LIN {X 0.030,Y -214.228,Z 1696.200,A 0.000,B 0.000,C 90.000,E1 35.931} C_DIS
LIN {X -0.002,Y -206.869,Z 1696.182,A 0.000,B 0.000,C 90.000,E1 32.801} C_DIS
LIN {X -0.016,Y -200.168,Z 1696.165,A 0.000,B 0.000,C 90.000,E1 29.617} C_DIS
LIN {X 0.061,Y -194.075,Z 1696.146,A 0.000,B 0.000,C 90.000,E1 26.360} C_DIS
LIN {X 0.072,Y -188.561,Z 1696.128,A 0.000,B 0.000,C 90.000,E1 23.078} C_DIS
LIN {X 0.078,Y -183.619,Z 1696.110,A 0.000,B 0.000,C 90.000,E1 19.758} C_DIS
LIN {X -0.045,Y -179.365,Z 1696.091,A 0.000,B 0.000,C 90.000,E1 16.441} C_DIS
LIN {X -0.073,Y -175.796,Z 1696.072,A 0.000,B 0.000,C 90.000,E1 13.063} C_DIS
LIN {X -0.080,Y -171.726,Z 1696.044,A 0.000,B 0.000,C 90.000,E1 7.936} C_DIS
LIN {X -0.053,Y -168.927,Z 1696.015,A 0.000,B 0.000,C 90.000,E1 2.751} C_DIS
LIN {X 0.075,Y -168.953,Z 1695.925,A 0.000,B 0.000,C 90.000,E1 346.464} C_DIS
LIN {X 0.065,Y -171.633,Z 1695.896,A 0.000,B 0.000,C 90.000,E1 341.275} C_DIS
LIN {X 0.068,Y -175.125,Z 1695.872,A 0.000,B 0.000,C 90.000,E1 336.975} C_DIS
LIN {X -0.029,Y -179.735,Z 1695.849,A 0.000,B 0.000,C 90.000,E1 332.743} C_DIS
LIN {X 0.084,Y -184.287,Z 1695.830,A 0.000,B 0.000,C 90.000,E1 329.331} C_DIS
LIN {X 0.045,Y -188.356,Z 1695.816,A 0.000,B 0.000,C 90.000,E1 326.834} C_DIS
LIN {X -0.013,Y -194.798,Z 1695.797,A 0.000,B 0.000,C 90.000,E1 323.543} C_DIS
LIN {X 0.017,Y -201.344,Z 1695.782,A 0.000,B 0.000,C 90.000,E1 320.678} C_DIS
LIN {X -0.010,Y -208.807,Z 1695.766,A 0.000,B 0.000,C 90.000,E1 317.877} C_DIS
LIN {X 0.119,Y -217.330,Z 1695.751,A 0.000,B 0.000,C 90.000,E1 315.081} C_DIS
LIN {X -0.014,Y -227.012,Z 1695.736,A 0.000,B 0.000,C 90.000,E1 312.405} C_DIS
LIN {X 0.124,Y -236.194,Z 1695.723,A 0.000,B 0.000,C 90.000,E1 310.092} C_DIS
LIN {X -0.018,Y -246.606,Z 1695.710,A 0.000,B 0.000,C 90.000,E1 307.890} C_DIS
LIN {X -0.140,Y -256.208,Z 1695.700,A 0.000,B 0.000,C 90.000,E1 306.091} C_DIS
LIN {X -0.025,Y -273.225,Z 1695.684,A 0.000,B 0.000,C 90.000,E1 303.214} C_DIS
LIN {X -0.060,Y -291.925,Z 1695.669,A 0.000,B 0.000,C 90.000,E1 300.463} C_DIS
LIN {X 0.104,Y -311.752,Z 1695.654,A 0.000,B 0.000,C 90.000,E1 297.769} C_DIS
LIN {X 0.030,Y -326.865,Z 1695.644,A 0.000,B 0.000,C 90.000,E1 295.848} C_DIS
LIN {X 0.100,Y -342.113,Z 1695.633,A 0.000,B 0.000,C 90.000,E1 293.951} C_DIS
LIN {X -0.138,Y -357.480,Z 1695.623,A 0.000,B 0.000,C 90.000,E1 292.153} C_DIS
LIN {X 0.084,Y -367.403,Z 1695.616,A 0.000,B 0.000,C 90.000,E1 290.918} C_DIS
LIN {X -0.082,Y -374.465,Z 1695.611,A 0.000,B 0.000,C 90.000,E1 290.066} C_DIS
LIN {X 0.242,Y -381.087,Z 1695.607,A 0.000,B 0.000,C 90.000,E1 289.141} C_DIS
LIN {X 0.012,Y -387.016,Z 1695.602,A 0.000,B 0.000,C 90.000,E1 288.308} C_DIS
LIN {X -0.191,Y -390.463,Z 1695.599,A 0.000,B 0.000,C 90.000,E1 287.764} C_DIS
LIN {X 0.165,Y -394.822,Z 1695.594,A 0.000,B 0.000,C 90.000,E1 286.858} C_DIS
LIN {X 0.065,Y -398.245,Z 1695.589,A 0.000,B 0.000,C 90.000,E1 286.024} C_DIS
LIN {X -0.074,Y -400.085,Z 1695.586,A 0.000,B 0.000,C 90.000,E1 285.481} C_DIS
LIN {X 0.072,Y -401.550,Z 1695.583,A 0.000,B 0.000,C 90.000,E1 284.898} C_DIS
LIN {X -0.054,Y -402.648,Z 1695.580,A 0.000,B 0.000,C 90.000,E1 284.356} C_DIS
LIN {X 0.117,Y -403.347,Z 1695.577,A 0.000,B 0.000,C 90.000,E1 283.772} C_DIS
LIN {X -0.094,Y -403.638,Z 1695.573,A 0.000,B 0.000,C 90.000,E1 283.244} C_DIS
LIN {X 0.182,Y -403.524,Z 1695.570,A 0.000,B 0.000,C 90.000,E1 282.647} C_DIS
LIN {X -0.024,Y -402.949,Z 1695.567,A 0.000,B 0.000,C 90.000,E1 282.119} C_DIS
LIN {X 0.163,Y -401.886,Z 1695.564,A 0.000,B 0.000,C 90.000,E1 281.535} C_DIS
LIN {X -0.048,Y -400.295,Z 1695.561,A 0.000,B 0.000,C 90.000,E1 281.007} C_DIS
LIN {X 0.055,Y -398.253,Z 1695.558,A 0.000,B 0.000,C 90.000,E1 280.433} C_DIS
LIN {X -0.169,Y -395.628,Z 1695.555,A 0.000,B 0.000,C 90.000,E1 279.905} C_DIS
LIN {X 0.037,Y -390.912,Z 1695.550,A 0.000,B 0.000,C 90.000,E1 279.029} C_DIS
LIN {X 0.178,Y -383.721,Z 1695.544,A 0.000,B 0.000,C 90.000,E1 277.871} C_DIS
LIN {X -0.205,Y -377.617,Z 1695.539,A 0.000,B 0.000,C 90.000,E1 277.068} C_DIS
LIN {X 0.194,Y -372.861,Z 1695.536,A 0.000,B 0.000,C 90.000,E1 276.429} C_DIS
LIN {X 0.146,Y -367.523,Z 1695.533,A 0.000,B 0.000,C 90.000,E1 275.853} C_DIS
LIN {X -0.105,Y -361.689,Z 1695.530,A 0.000,B 0.000,C 90.000,E1 275.334} C_DIS
LIN {X -0.096,Y -355.702,Z 1695.527,A 0.000,B 0.000,C 90.000,E1 274.821} C_DIS
LIN {X -0.140,Y -349.396,Z 1695.524,A 0.000,B 0.000,C 90.000,E1 274.359} C_DIS
LIN {X -0.004,Y -339.856,Z 1695.521,A 0.000,B 0.000,C 90.000,E1 273.726} C_DIS
LIN {X -0.104,Y -329.964,Z 1695.518,A 0.000,B 0.000,C 90.000,E1 273.212} C_DIS
LIN {X -0.070,Y -320.129,Z 1695.515,A 0.000,B 0.000,C 90.000,E1 272.751} C_DIS
LIN {X -0.097,Y -309.761,Z 1695.513,A 0.000,B 0.000,C 90.000,E1 272.350} C_DIS
LIN {X 0.055,Y -296.182,Z 1695.511,A 0.000,B 0.000,C 90.000,E1 271.892} C_DIS
LIN {X 0.143,Y -285.442,Z 1695.509,A 0.000,B 0.000,C 90.000,E1 271.604} C_DIS
LIN {X -0.086,Y -273.014,Z 1695.508,A 0.000,B 0.000,C 90.000,E1 271.432} C_DIS
LIN {X -0.108,Y -263.030,Z 1695.507,A 0.000,B 0.000,C 90.000,E1 271.318} C_DIS
LIN {X 0.113,Y -249.683,Z 1695.507,A 0.000,B 0.000,C 90.000,E1 271.203} C_DIS
LIN {X 0.064,Y -190.443,Z 1695.507,A 0.000,B 0.000,C 90.000,E1 271.203} C_DIS
LIN {X -0.003,Y -184.503,Z 1695.507,A 0.000,B 0.000,C 90.000,E1 271.203} C_DIS
LIN {X -0.024,Y -181.413,Z 1695.507,A 0.000,B 0.000,C 90.000,E1 271.203} C_DIS
LIN {X 0.029,Y -181.579,Z 1695.501,A 0.000,B 0.000,C 90.000,E1 270.172} C_DIS
LIN {X 0.033,Y -180.853,Z 1695.472,A 0.000,B 0.000,C 90.000,E1 264.951} C_DIS
LIN {X -0.062,Y -178.964,Z 1695.444,A 0.000,B 0.000,C 90.000,E1 259.916} C_DIS
LIN {X 0.006,Y -177.372,Z 1695.430,A 0.000,B 0.000,C 90.000,E1 257.353} C_DIS
LIN {X -0.067,Y -175.547,Z 1695.411,A 0.000,B 0.000,C 90.000,E1 253.976} C_DIS
LIN {X -0.059,Y -172.279,Z 1695.387,A 0.000,B 0.000,C 90.000,E1 249.699} C_DIS
LIN {X -0.020,Y -171.758,Z 1695.382,A 0.000,B 0.000,C 90.000,E1 248.827} C_DIS
LIN {X -0.003,Y -167.358,Z 1695.354,A 0.000,B 0.000,C 90.000,E1 243.640} C_DIS
LIN {X 0.080,Y -166.747,Z 1695.349,A 0.000,B 0.000,C 90.000,E1 242.743} C_DIS
LIN {X -0.009,Y -162.727,Z 1695.324,A 0.000,B 0.000,C 90.000,E1 238.408} C_DIS
LIN {X 0.052,Y -161.417,Z 1695.315,A 0.000,B 0.000,C 90.000,E1 236.628} C_DIS
LIN {X 0.094,Y -157.409,Z 1695.290,A 0.000,B 0.000,C 90.000,E1 232.190} C_DIS
LIN {X 0.027,Y -155.411,Z 1695.275,A 0.000,B 0.000,C 90.000,E1 229.542} C_DIS
LIN {X -0.042,Y -151.740,Z 1695.250,A 0.000,B 0.000,C 90.000,E1 225.081} C_DIS
LIN {X -0.030,Y -149.937,Z 1695.235,A 0.000,B 0.000,C 90.000,E1 222.366} C_DIS
LIN {X -0.002,Y -146.785,Z 1695.210,A 0.000,B 0.000,C 90.000,E1 217.810} C_DIS
LIN {X -0.018,Y -145.357,Z 1695.195,A 0.000,B 0.000,C 90.000,E1 215.072} C_DIS
LIN {X 0.016,Y -142.427,Z 1695.164,A 0.000,B 0.000,C 90.000,E1 209.539} C_DIS
LIN {X 0.064,Y -141.415,Z 1695.149,A 0.000,B 0.000,C 90.000,E1 206.744} C_DIS
LIN {X 0.052,Y -139.361,Z 1695.113,A 0.000,B 0.000,C 90.000,E1 200.248} C_DIS
LIN {X 0.039,Y -138.803,Z 1695.097,A 0.000,B 0.000,C 90.000,E1 197.457} C_DIS
LIN {X -0.042,Y -138.349,Z 1695.056,A 0.000,B 0.000,C 90.000,E1 190.018} C_DIS
LIN {X -0.027,Y -139.365,Z 1695.009,A 0.000,B 0.000,C 90.000,E1 181.604} C_DIS
LIN {X 0.026,Y -141.250,Z 1694.973,A 0.000,B 0.000,C 90.000,E1 175.065} C_DIS
LIN {X -0.016,Y -142.619,Z 1694.957,A 0.000,B 0.000,C 90.000,E1 172.299} C_DIS
LIN {X -0.063,Y -144.938,Z 1694.932,A 0.000,B 0.000,C 90.000,E1 167.701} C_DIS
LIN {X 0.070,Y -147.566,Z 1694.911,A 0.000,B 0.000,C 90.000,E1 163.976} C_DIS
LIN {X -0.040,Y -150.174,Z 1694.891,A 0.000,B 0.000,C 90.000,E1 160.369} C_DIS
LIN {X -0.032,Y -153.551,Z 1694.871,A 0.000,B 0.000,C 90.000,E1 156.741} C_DIS
LIN {X 0.020,Y -156.968,Z 1694.851,A 0.000,B 0.000,C 90.000,E1 153.127} C_DIS
LIN {X -0.045,Y -161.077,Z 1694.831,A 0.000,B 0.000,C 90.000,E1 149.587} C_DIS
LIN {X 0.040,Y -163.184,Z 1694.821,A 0.000,B 0.000,C 90.000,E1 147.788} C_DIS
LIN {X 0.046,Y -167.605,Z 1694.802,A 0.000,B 0.000,C 90.000,E1 144.276} C_DIS
LIN {X -0.045,Y -171.433,Z 1694.787,A 0.000,B 0.000,C 90.000,E1 141.698} C_DIS
LIN {X -0.007,Y -176.354,Z 1694.768,A 0.000,B 0.000,C 90.000,E1 138.243} C_DIS
LIN {X -0.011,Y -180.645,Z 1694.754,A 0.000,B 0.000,C 90.000,E1 135.688} C_DIS
LIN {X -0.026,Y -186.047,Z 1694.735,A 0.000,B 0.000,C 90.000,E1 132.324} C_DIS
LIN {X 0.036,Y -190.683,Z 1694.721,A 0.000,B 0.000,C 90.000,E1 129.806} C_DIS
LIN {X 0.069,Y -196.434,Z 1694.703,A 0.000,B 0.000,C 90.000,E1 126.503} C_DIS
LIN {X 0.037,Y -201.219,Z 1694.689,A 0.000,B 0.000,C 90.000,E1 124.072} C_DIS
LIN {X 0.048,Y -207.544,Z 1694.670,A 0.000,B 0.000,C 90.000,E1 120.669} C_DIS
LIN {X 0.007,Y -208.682,Z 1694.667,A 0.000,B 0.000,C 90.000,E1 120.129} C_DIS
LIN {X -0.025,Y -331.531,Z 1694.667,A 0.000,B 0.000,C 90.000,E1 120.129} C_DIS
LIN {X -0.066,Y -334.422,Z 1694.667,A 0.000,B 0.000,C 90.000,E1 120.079} C_DIS
LIN {X 0.082,Y -337.325,Z 1694.666,A 0.000,B 0.000,C 90.000,E1 119.922} C_DIS
LIN {X -0.059,Y -340.923,Z 1694.665,A 0.000,B 0.000,C 90.000,E1 119.667} C_DIS
LIN {X 0.003,Y -344.532,Z 1694.662,A 0.000,B 0.000,C 90.000,E1 119.205} C_DIS
LIN {X -0.009,Y -346.257,Z 1694.661,A 0.000,B 0.000,C 90.000,E1 118.899} C_DIS
LIN {X 0.097,Y -360.412,Z 1694.644,A 0.000,B 0.000,C 90.000,E1 115.848} C_DIS
LIN {X -0.077,Y -374.699,Z 1694.629,A 0.000,B 0.000,C 90.000,E1 113.206} C_DIS
LIN {X 0.067,Y -388.768,Z 1694.616,A 0.000,B 0.000,C 90.000,E1 110.865} C_DIS
LIN {X 0.061,Y -404.224,Z 1694.603,A 0.000,B 0.000,C 90.000,E1 108.598} C_DIS
LIN {X 0.046,Y -421.177,Z 1694.591,A 0.000,B 0.000,C 90.000,E1 106.386} C_DIS
LIN {X -0.074,Y -439.740,Z 1694.579,A 0.000,B 0.000,C 90.000,E1 104.245} C_DIS
LIN {X -0.046,Y -459.590,Z 1694.568,A 0.000,B 0.000,C 90.000,E1 102.187} C_DIS
LIN {X -0.042,Y -482.573,Z 1694.556,A 0.000,B 0.000,C 90.000,E1 100.074} C_DIS
LIN {X 0.077,Y -503.529,Z 1694.546,A 0.000,B 0.000,C 90.000,E1 98.341} C_DIS
LIN {X -0.170,Y -505.736,Z 1694.545,A 0.000,B 0.000,C 90.000,E1 98.163} C_DIS
LIN {X -0.204,Y -507.593,Z 1694.544,A 0.000,B 0.000,C 90.000,E1 97.936} C_DIS
LIN {X -0.168,Y -508.999,Z 1694.543,A 0.000,B 0.000,C 90.000,E1 97.701} C_DIS
LIN {X 0.164,Y -510.872,Z 1694.540,A 0.000,B 0.000,C 90.000,E1 97.182} C_DIS
LIN {X 0.000,Y -511.603,Z 1694.537,A 0.000,B 0.000,C 90.000,E1 96.720} C_DIS
LIN {X -0.155,Y -511.316,Z 1694.535,A 0.000,B 0.000,C 90.000,E1 96.258} C_DIS
LIN {X 0.201,Y -509.964,Z 1694.532,A 0.000,B 0.000,C 90.000,E1 95.739} C_DIS
LIN {X 0.100,Y -508.818,Z 1694.531,A 0.000,B 0.000,C 90.000,E1 95.511} C_DIS
LIN {X -0.059,Y -505.504,Z 1694.528,A 0.000,B 0.000,C 90.000,E1 95.049} C_DIS
LIN {X -0.182,Y -494.848,Z 1694.520,A 0.000,B 0.000,C 90.000,E1 93.612} C_DIS
LIN {X -0.020,Y -484.051,Z 1694.512,A 0.000,B 0.000,C 90.000,E1 92.121} C_DIS
LIN {X -0.222,Y -471.379,Z 1694.502,A 0.000,B 0.000,C 90.000,E1 90.401} C_DIS
LIN {X 0.000,Y -460.498,Z 1694.494,A 0.000,B 0.000,C 90.000,E1 88.854} C_DIS
LIN {X 0.036,Y -449.452,Z 1694.485,A 0.000,B 0.000,C 90.000,E1 87.306} C_DIS
LIN {X -0.089,Y -438.224,Z 1694.476,A 0.000,B 0.000,C 90.000,E1 85.755} C_DIS
LIN {X 0.191,Y -424.959,Z 1694.466,A 0.000,B 0.000,C 90.000,E1 83.856} C_DIS
LIN {X 0.022,Y -408.389,Z 1694.452,A 0.000,B 0.000,C 90.000,E1 81.432} C_DIS
LIN {X 0.199,Y -387.530,Z 1694.434,A 0.000,B 0.000,C 90.000,E1 78.049} C_DIS
LIN {X 0.168,Y -374.325,Z 1694.421,A 0.000,B 0.000,C 90.000,E1 75.755} C_DIS
LIN {X 0.016,Y -361.481,Z 1694.408,A 0.000,B 0.000,C 90.000,E1 73.433} C_DIS
LIN {X 0.064,Y -345.943,Z 1694.391,A 0.000,B 0.000,C 90.000,E1 70.423} C_DIS
LIN {X -0.014,Y -331.397,Z 1694.374,A 0.000,B 0.000,C 90.000,E1 67.358} C_DIS
LIN {X -0.093,Y -318.829,Z 1694.358,A 0.000,B 0.000,C 90.000,E1 64.537} C_DIS
LIN {X -0.097,Y -306.555,Z 1694.342,A 0.000,B 0.000,C 90.000,E1 61.641} C_DIS
LIN {X -0.046,Y -298.534,Z 1694.331,A 0.000,B 0.000,C 90.000,E1 59.665} C_DIS
LIN {X -0.009,Y -288.988,Z 1694.318,A 0.000,B 0.000,C 90.000,E1 57.327} C_DIS
LIN {X -0.069,Y -280.700,Z 1694.307,A 0.000,B 0.000,C 90.000,E1 55.308} C_DIS
LIN {X 0.104,Y -272.100,Z 1694.296,A 0.000,B 0.000,C 90.000,E1 53.210} C_DIS
LIN {X -0.089,Y -262.186,Z 1694.282,A 0.000,B 0.000,C 90.000,E1 50.803} C_DIS
LIN {X 0.009,Y -252.457,Z 1694.268,A 0.000,B 0.000,C 90.000,E1 48.286} C_DIS
LIN {X 0.037,Y -240.583,Z 1694.250,A 0.000,B 0.000,C 90.000,E1 45.000} C_DIS
LIN {X -0.055,Y -230.918,Z 1694.234,A 0.000,B 0.000,C 90.000,E1 42.043} C_DIS
LIN {X -0.002,Y -222.030,Z 1694.217,A 0.000,B 0.000,C 90.000,E1 38.991} C_DIS
LIN {X 0.072,Y -214.005,Z 1694.199,A 0.000,B 0.000,C 90.000,E1 35.884} C_DIS
LIN {X 0.041,Y -206.678,Z 1694.182,A 0.000,B 0.000,C 90.000,E1 32.752} C_DIS
LIN {X -0.048,Y -200.026,Z 1694.164,A 0.000,B 0.000,C 90.000,E1 29.589} C_DIS
LIN {X -0.070,Y -193.968,Z 1694.146,A 0.000,B 0.000,C 90.000,E1 26.360} C_DIS
LIN {X -0.058,Y -188.449,Z 1694.128,A 0.000,B 0.000,C 90.000,E1 23.078} C_DIS
LIN {X -0.052,Y -183.528,Z 1694.110,A 0.000,B 0.000,C 90.000,E1 19.758} C_DIS
LIN {X -0.001,Y -179.277,Z 1694.091,A 0.000,B 0.000,C 90.000,E1 16.386} C_DIS
LIN {X -0.030,Y -175.708,Z 1694.072,A 0.000,B 0.000,C 90.000,E1 13.008} C_DIS
LIN {X -0.064,Y -172.241,Z 1694.048,A 0.000,B 0.000,C 90.000,E1 8.746} C_DIS
LIN {X -0.002,Y -169.206,Z 1694.020,A 0.000,B 0.000,C 90.000,E1 3.555} C_DIS
LIN {X 0.014,Y -167.284,Z 1693.973,A 0.000,B 0.000,C 90.000,E1 355.179} C_DIS
LIN {X 0.070,Y -168.897,Z 1693.925,A 0.000,B 0.000,C 90.000,E1 346.464} C_DIS
LIN {X 0.056,Y -171.617,Z 1693.896,A 0.000,B 0.000,C 90.000,E1 341.275} C_DIS
LIN {X 0.059,Y -175.114,Z 1693.872,A 0.000,B 0.000,C 90.000,E1 336.975} C_DIS
LIN {X -0.038,Y -179.765,Z 1693.849,A 0.000,B 0.000,C 90.000,E1 332.743} C_DIS
LIN {X 0.076,Y -184.359,Z 1693.830,A 0.000,B 0.000,C 90.000,E1 329.331} C_DIS
LIN {X 0.037,Y -188.457,Z 1693.816,A 0.000,B 0.000,C 90.000,E1 326.834} C_DIS
LIN {X -0.018,Y -194.926,Z 1693.797,A 0.000,B 0.000,C 90.000,E1 323.543} C_DIS
LIN {X 0.015,Y -201.480,Z 1693.782,A 0.000,B 0.000,C 90.000,E1 320.678} C_DIS
LIN {X -0.009,Y -208.972,Z 1693.766,A 0.000,B 0.000,C 90.000,E1 317.877} C_DIS
LIN {X -0.030,Y -217.522,Z 1693.751,A 0.000,B 0.000,C 90.000,E1 315.121} C_DIS
LIN {X -0.005,Y -227.218,Z 1693.736,A 0.000,B 0.000,C 90.000,E1 312.405} C_DIS
LIN {X 0.138,Y -236.411,Z 1693.723,A 0.000,B 0.000,C 90.000,E1 310.092} C_DIS
LIN {X 0.001,Y -246.816,Z 1693.710,A 0.000,B 0.000,C 90.000,E1 307.890} C_DIS
LIN {X -0.117,Y -256.413,Z 1693.700,A 0.000,B 0.000,C 90.000,E1 306.091} C_DIS
LIN {X 0.004,Y -273.378,Z 1693.685,A 0.000,B 0.000,C 90.000,E1 303.214} C_DIS
LIN {X -0.025,Y -292.060,Z 1693.669,A 0.000,B 0.000,C 90.000,E1 300.463} C_DIS
LIN {X 0.145,Y -311.848,Z 1693.654,A 0.000,B 0.000,C 90.000,E1 297.769} C_DIS
LIN {X 0.075,Y -326.940,Z 1693.644,A 0.000,B 0.000,C 90.000,E1 295.848} C_DIS
LIN {X 0.148,Y -342.149,Z 1693.633,A 0.000,B 0.000,C 90.000,E1 293.951} C_DIS
LIN {X -0.088,Y -357.514,Z 1693.623,A 0.000,B 0.000,C 90.000,E1 292.153} C_DIS
LIN {X 0.137,Y -367.416,Z 1693.616,A 0.000,B 0.000,C 90.000,E1 290.918} C_DIS
LIN {X -0.092,Y -374.554,Z 1693.611,A 0.000,B 0.000,C 90.000,E1 290.066} C_DIS
LIN {X 0.232,Y -381.182,Z 1693.607,A 0.000,B 0.000,C 90.000,E1 289.141} C_DIS
LIN {X 0.004,Y -387.101,Z 1693.602,A 0.000,B 0.000,C 90.000,E1 288.308} C_DIS
LIN {X -0.199,Y -390.540,Z 1693.599,A 0.000,B 0.000,C 90.000,E1 287.764} C_DIS
LIN {X 0.157,Y -394.932,Z 1693.594,A 0.000,B 0.000,C 90.000,E1 286.858} C_DIS
LIN {X 0.059,Y -398.389,Z 1693.589,A 0.000,B 0.000,C 90.000,E1 286.024} C_DIS
LIN {X -0.080,Y -400.222,Z 1693.586,A 0.000,B 0.000,C 90.000,E1 285.481} C_DIS
LIN {X 0.067,Y -401.679,Z 1693.583,A 0.000,B 0.000,C 90.000,E1 284.898} C_DIS
LIN {X -0.059,Y -402.830,Z 1693.580,A 0.000,B 0.000,C 90.000,E1 284.356} C_DIS
LIN {X 0.114,Y -403.515,Z 1693.577,A 0.000,B 0.000,C 90.000,E1 283.772} C_DIS
LIN {X -0.096,Y -403.833,Z 1693.573,A 0.000,B 0.000,C 90.000,E1 283.244} C_DIS
LIN {X 0.182,Y -403.732,Z 1693.570,A 0.000,B 0.000,C 90.000,E1 282.647} C_DIS
LIN {X -0.024,Y -403.154,Z 1693.567,A 0.000,B 0.000,C 90.000,E1 282.119} C_DIS
LIN {X 0.164,Y -402.104,Z 1693.564,A 0.000,B 0.000,C 90.000,E1 281.535} C_DIS
LIN {X -0.046,Y -400.527,Z 1693.561,A 0.000,B 0.000,C 90.000,E1 281.007} C_DIS
LIN {X 0.058,Y -398.464,Z 1693.558,A 0.000,B 0.000,C 90.000,E1 280.433} C_DIS
LIN {X -0.165,Y -395.866,Z 1693.555,A 0.000,B 0.000,C 90.000,E1 279.905} C_DIS
LIN {X 0.044,Y -391.171,Z 1693.550,A 0.000,B 0.000,C 90.000,E1 279.029} C_DIS
LIN {X 0.150,Y -385.815,Z 1693.545,A 0.000,B 0.000,C 90.000,E1 278.163} C_DIS
LIN {X -0.175,Y -379.906,Z 1693.541,A 0.000,B 0.000,C 90.000,E1 277.352} C_DIS
LIN {X -0.178,Y -375.435,Z 1693.537,A 0.000,B 0.000,C 90.000,E1 276.777} C_DIS
LIN {X 0.164,Y -370.366,Z 1693.534,A 0.000,B 0.000,C 90.000,E1 276.144} C_DIS
LIN {X -0.150,Y -364.742,Z 1693.531,A 0.000,B 0.000,C 90.000,E1 275.625} C_DIS
LIN {X 0.139,Y -358.847,Z 1693.528,A 0.000,B 0.000,C 90.000,E1 275.049} C_DIS
LIN {X -0.023,Y -352.666,Z 1693.526,A 0.000,B 0.000,C 90.000,E1 274.588} C_DIS
LIN {X 0.048,Y -346.231,Z 1693.523,A 0.000,B 0.000,C 90.000,E1 274.131} C_DIS
LIN {X 0.067,Y -339.748,Z 1693.521,A 0.000,B 0.000,C 90.000,E1 273.726} C_DIS
LIN {X -0.040,Y -329.761,Z 1693.518,A 0.000,B 0.000,C 90.000,E1 273.212} C_DIS
LIN {X -0.023,Y -319.765,Z 1693.515,A 0.000,B 0.000,C 90.000,E1 272.751} C_DIS
LIN {X 0.050,Y -313.001,Z 1693.514,A 0.000,B 0.000,C 90.000,E1 272.465} C_DIS
LIN {X -0.019,Y -302.463,Z 1693.512,A 0.000,B 0.000,C 90.000,E1 272.121} C_DIS
LIN {X -0.068,Y -292.250,Z 1693.510,A 0.000,B 0.000,C 90.000,E1 271.835} C_DIS
LIN {X 0.100,Y -280.775,Z 1693.509,A 0.000,B 0.000,C 90.000,E1 271.547} C_DIS
LIN {X -0.023,Y -268.128,Z 1693.508,A 0.000,B 0.000,C 90.000,E1 271.375} C_DIS
LIN {X 0.128,Y -259.488,Z 1693.507,A 0.000,B 0.000,C 90.000,E1 271.260} C_DIS
LIN {X -0.001,Y -250.689,Z 1693.507,A 0.000,B 0.000,C 90.000,E1 271.260} C_DIS
LIN {X -0.023,Y -196.001,Z 1693.507,A 0.000,B 0.000,C 90.000,E1 271.260} C_DIS
LIN {X 0.038,Y -186.326,Z 1693.507,A 0.000,B 0.000,C 90.000,E1 271.203} C_DIS
LIN {X 0.001,Y -181.411,Z 1693.507,A 0.000,B 0.000,C 90.000,E1 271.203} C_DIS
LIN {X -0.015,Y -181.581,Z 1693.502,A 0.000,B 0.000,C 90.000,E1 270.286} C_DIS
LIN {X -0.040,Y -180.899,Z 1693.474,A 0.000,B 0.000,C 90.000,E1 265.241} C_DIS
LIN {X -0.091,Y -180.211,Z 1693.464,A 0.000,B 0.000,C 90.000,E1 263.571} C_DIS
LIN {X 0.039,Y -179.033,Z 1693.445,A 0.000,B 0.000,C 90.000,E1 260.151} C_DIS
LIN {X -0.074,Y -178.686,Z 1693.441,A 0.000,B 0.000,C 90.000,E1 259.342} C_DIS
LIN {X 0.037,Y -175.736,Z 1693.412,A 0.000,B 0.000,C 90.000,E1 254.212} C_DIS
LIN {X 0.033,Y -171.920,Z 1693.384,A 0.000,B 0.000,C 90.000,E1 249.082} C_DIS
LIN {X 0.007,Y -171.291,Z 1693.379,A 0.000,B 0.000,C 90.000,E1 248.230} C_DIS
LIN {X 0.053,Y -167.556,Z 1693.355,A 0.000,B 0.000,C 90.000,E1 243.896} C_DIS
LIN {X 0.067,Y -166.179,Z 1693.345,A 0.000,B 0.000,C 90.000,E1 242.153} C_DIS
LIN {X 0.056,Y -162.950,Z 1693.326,A 0.000,B 0.000,C 90.000,E1 238.663} C_DIS
LIN {X 0.103,Y -160.856,Z 1693.311,A 0.000,B 0.000,C 90.000,E1 236.008} C_DIS
LIN {X 0.081,Y -157.633,Z 1693.292,A 0.000,B 0.000,C 90.000,E1 232.477} C_DIS
LIN {X 0.018,Y -155.670,Z 1693.277,A 0.000,B 0.000,C 90.000,E1 229.828} C_DIS
LIN {X 0.071,Y -151.937,Z 1693.252,A 0.000,B 0.000,C 90.000,E1 225.324} C_DIS
LIN {X 0.085,Y -150.175,Z 1693.237,A 0.000,B 0.000,C 90.000,E1 222.609} C_DIS
LIN {X 0.005,Y -146.951,Z 1693.212,A 0.000,B 0.000,C 90.000,E1 218.096} C_DIS
LIN {X -0.007,Y -145.538,Z 1693.196,A 0.000,B 0.000,C 90.000,E1 215.358} C_DIS
LIN {X 0.031,Y -142.935,Z 1693.171,A 0.000,B 0.000,C 90.000,E1 210.747} C_DIS
LIN {X -0.033,Y -141.558,Z 1693.150,A 0.000,B 0.000,C 90.000,E1 207.078} C_DIS
LIN {X 0.020,Y -139.408,Z 1693.114,A 0.000,B 0.000,C 90.000,E1 200.556} C_DIS
LIN {X -0.059,Y -139.128,Z 1693.104,A 0.000,B 0.000,C 90.000,E1 198.725} C_DIS
LIN {X -0.032,Y -138.350,Z 1693.057,A 0.000,B 0.000,C 90.000,E1 190.310} C_DIS
LIN {X -0.044,Y -139.498,Z 1693.005,A 0.000,B 0.000,C 90.000,E1 180.974} C_DIS
LIN {X 0.037,Y -141.121,Z 1692.974,A 0.000,B 0.000,C 90.000,E1 175.355} C_DIS
LIN {X -0.010,Y -142.502,Z 1692.959,A 0.000,B 0.000,C 90.000,E1 172.591} C_DIS
LIN {X -0.064,Y -144.757,Z 1692.933,A 0.000,B 0.000,C 90.000,E1 167.993} C_DIS
LIN {X 0.027,Y -147.368,Z 1692.913,A 0.000,B 0.000,C 90.000,E1 164.283} C_DIS
LIN {X -0.051,Y -150.696,Z 1692.887,A 0.000,B 0.000,C 90.000,E1 159.752} C_DIS
LIN {X 0.032,Y -154.175,Z 1692.867,A 0.000,B 0.000,C 90.000,E1 156.102} C_DIS
LIN {X -0.038,Y -157.611,Z 1692.847,A 0.000,B 0.000,C 90.000,E1 152.538} C_DIS
LIN {X 0.050,Y -161.863,Z 1692.828,A 0.000,B 0.000,C 90.000,E1 148.948} C_DIS
LIN {X -0.071,Y -166.054,Z 1692.808,A 0.000,B 0.000,C 90.000,E1 145.468} C_DIS
LIN {X -0.080,Y -171.059,Z 1692.789,A 0.000,B 0.000,C 90.000,E1 141.984} C_DIS
LIN {X -0.050,Y -175.931,Z 1692.770,A 0.000,B 0.000,C 90.000,E1 138.528} C_DIS
LIN {X -0.058,Y -180.170,Z 1692.755,A 0.000,B 0.000,C 90.000,E1 135.972} C_DIS
LIN {X -0.090,Y -185.587,Z 1692.737,A 0.000,B 0.000,C 90.000,E1 132.609} C_DIS
LIN {X -0.040,Y -190.178,Z 1692.723,A 0.000,B 0.000,C 90.000,E1 130.092} C_DIS
LIN {X 0.005,Y -197.508,Z 1692.700,A 0.000,B 0.000,C 90.000,E1 125.964} C_DIS
LIN {X 0.046,Y -200.776,Z 1692.691,A 0.000,B 0.000,C 90.000,E1 124.326} C_DIS
LIN {X -0.044,Y -206.667,Z 1692.673,A 0.000,B 0.000,C 90.000,E1 121.131} C_DIS
LIN {X -0.036,Y -208.602,Z 1692.668,A 0.000,B 0.000,C 90.000,E1 120.178} C_DIS
LIN {X 0.181,Y -331.416,Z 1692.668,A 0.000,B 0.000,C 90.000,E1 120.129} C_DIS
LIN {X 0.084,Y -332.682,Z 1692.667,A 0.000,B 0.000,C 90.000,E1 120.129} C_DIS
LIN {X -0.072,Y -336.857,Z 1692.667,A 0.000,B 0.000,C 90.000,E1 120.001} C_DIS
LIN {X 0.063,Y -339.147,Z 1692.666,A 0.000,B 0.000,C 90.000,E1 119.823} C_DIS
LIN {X -0.086,Y -342.286,Z 1692.664,A 0.000,B 0.000,C 90.000,E1 119.539} C_DIS
LIN {X -0.111,Y -345.841,Z 1692.661,A 0.000,B 0.000,C 90.000,E1 118.999} C_DIS
LIN {X -0.149,Y -361.491,Z 1692.642,A 0.000,B 0.000,C 90.000,E1 115.668} C_DIS
LIN {X 0.197,Y -375.906,Z 1692.628,A 0.000,B 0.000,C 90.000,E1 112.950} C_DIS
LIN {X 0.012,Y -390.096,Z 1692.615,A 0.000,B 0.000,C 90.000,E1 110.663} C_DIS
LIN {X -0.107,Y -405.685,Z 1692.602,A 0.000,B 0.000,C 90.000,E1 108.417} C_DIS
LIN {X -0.091,Y -422.779,Z 1692.590,A 0.000,B 0.000,C 90.000,E1 106.205} C_DIS
LIN {X -0.180,Y -441.497,Z 1692.578,A 0.000,B 0.000,C 90.000,E1 104.064} C_DIS
LIN {X -0.035,Y -461.400,Z 1692.567,A 0.000,B 0.000,C 90.000,E1 102.007} C_DIS
LIN {X 0.011,Y -484.436,Z 1692.555,A 0.000,B 0.000,C 90.000,E1 99.905} C_DIS
LIN {X 0.059,Y -502.801,Z 1692.547,A 0.000,B 0.000,C 90.000,E1 98.398} C_DIS
LIN {X -0.173,Y -505.121,Z 1692.546,A 0.000,B 0.000,C 90.000,E1 98.219} C_DIS
LIN {X 0.021,Y -506.880,Z 1692.544,A 0.000,B 0.000,C 90.000,E1 97.992} C_DIS
LIN {X -0.037,Y -508.464,Z 1692.543,A 0.000,B 0.000,C 90.000,E1 97.757} C_DIS
LIN {X -0.163,Y -509.645,Z 1692.542,A 0.000,B 0.000,C 90.000,E1 97.530} C_DIS
LIN {X 0.176,Y -511.052,Z 1692.539,A 0.000,B 0.000,C 90.000,E1 97.011} C_DIS
LIN {X 0.017,Y -511.389,Z 1692.536,A 0.000,B 0.000,C 90.000,E1 96.549} C_DIS
LIN {X -0.136,Y -510.711,Z 1692.534,A 0.000,B 0.000,C 90.000,E1 96.087} C_DIS
LIN {X 0.221,Y -508.900,Z 1692.531,A 0.000,B 0.000,C 90.000,E1 95.568} C_DIS
LIN {X 0.166,Y -507.457,Z 1692.530,A 0.000,B 0.000,C 90.000,E1 95.334} C_DIS
LIN {X -0.059,Y -495.068,Z 1692.520,A 0.000,B 0.000,C 90.000,E1 93.669} C_DIS
LIN {X 0.104,Y -484.289,Z 1692.512,A 0.000,B 0.000,C 90.000,E1 92.178} C_DIS
LIN {X -0.102,Y -471.624,Z 1692.502,A 0.000,B 0.000,C 90.000,E1 90.458} C_DIS
LIN {X 0.122,Y -460.741,Z 1692.494,A 0.000,B 0.000,C 90.000,E1 88.912} C_DIS
LIN {X 0.160,Y -449.733,Z 1692.485,A 0.000,B 0.000,C 90.000,E1 87.364} C_DIS
LIN {X 0.206,Y -436.612,Z 1692.475,A 0.000,B 0.000,C 90.000,E1 85.527} C_DIS
LIN {X 0.180,Y -421.443,Z 1692.463,A 0.000,B 0.000,C 90.000,E1 83.394} C_DIS
LIN {X -0.130,Y -406.764,Z 1692.451,A 0.000,B 0.000,C 90.000,E1 81.254} C_DIS
LIN {X -0.073,Y -385.987,Z 1692.433,A 0.000,B 0.000,C 90.000,E1 77.881} C_DIS
LIN {X -0.048,Y -372.788,Z 1692.420,A 0.000,B 0.000,C 90.000,E1 75.574} C_DIS
LIN {X 0.119,Y -359.960,Z 1692.407,A 0.000,B 0.000,C 90.000,E1 73.196} C_DIS
LIN {X 0.112,Y -344.472,Z 1692.390,A 0.000,B 0.000,C 90.000,E1 70.188} C_DIS
LIN {X 0.126,Y -331.422,Z 1692.375,A 0.000,B 0.000,C 90.000,E1 67.411} C_DIS
LIN {X 0.054,Y -318.860,Z 1692.359,A 0.000,B 0.000,C 90.000,E1 64.588} C_DIS
LIN {X 0.048,Y -306.589,Z 1692.343,A 0.000,B 0.000,C 90.000,E1 61.691} C_DIS
LIN {X -0.050,Y -298.566,Z 1692.332,A 0.000,B 0.000,C 90.000,E1 59.744} C_DIS
LIN {X 0.145,Y -289.028,Z 1692.319,A 0.000,B 0.000,C 90.000,E1 57.375} C_DIS
LIN {X -0.073,Y -280.721,Z 1692.308,A 0.000,B 0.000,C 90.000,E1 55.388} C_DIS
LIN {X -0.121,Y -272.130,Z 1692.296,A 0.000,B 0.000,C 90.000,E1 53.336} C_DIS
LIN {X -0.040,Y -260.777,Z 1692.281,A 0.000,B 0.000,C 90.000,E1 50.517} C_DIS
LIN {X 0.024,Y -251.064,Z 1692.267,A 0.000,B 0.000,C 90.000,E1 48.000} C_DIS
LIN {X 0.006,Y -239.326,Z 1692.248,A 0.000,B 0.000,C 90.000,E1 44.717} C_DIS
LIN {X -0.001,Y -228.651,Z 1692.230,A 0.000,B 0.000,C 90.000,E1 41.353} C_DIS
LIN {X 0.071,Y -221.026,Z 1692.215,A 0.000,B 0.000,C 90.000,E1 38.669} C_DIS
LIN {X -0.015,Y -213.117,Z 1692.198,A 0.000,B 0.000,C 90.000,E1 35.598} C_DIS
LIN {X -0.068,Y -205.886,Z 1692.180,A 0.000,B 0.000,C 90.000,E1 32.467} C_DIS
LIN {X -0.102,Y -199.321,Z 1692.162,A 0.000,B 0.000,C 90.000,E1 29.283} C_DIS
LIN {X -0.047,Y -193.335,Z 1692.145,A 0.000,B 0.000,C 90.000,E1 26.027} C_DIS
LIN {X 0.043,Y -187.880,Z 1692.126,A 0.000,B 0.000,C 90.000,E1 22.717} C_DIS
LIN {X 0.036,Y -183.036,Z 1692.108,A 0.000,B 0.000,C 90.000,E1 19.396} C_DIS
LIN {X 0.073,Y -178.843,Z 1692.089,A 0.000,B 0.000,C 90.000,E1 16.024} C_DIS
LIN {X 0.028,Y -175.347,Z 1692.070,A 0.000,B 0.000,C 90.000,E1 12.647} C_DIS
LIN {X -0.054,Y -171.950,Z 1692.047,A 0.000,B 0.000,C 90.000,E1 8.398} C_DIS
LIN {X -0.018,Y -168.990,Z 1692.018,A 0.000,B 0.000,C 90.000,E1 3.212} C_DIS
LIN {X 0.013,Y -167.228,Z 1691.973,A 0.000,B 0.000,C 90.000,E1 355.179} C_DIS
LIN {X 0.064,Y -168.855,Z 1691.925,A 0.000,B 0.000,C 90.000,E1 346.464} C_DIS
LIN {X 0.049,Y -171.597,Z 1691.896,A 0.000,B 0.000,C 90.000,E1 341.275} C_DIS
LIN {X 0.051,Y -175.105,Z 1691.872,A 0.000,B 0.000,C 90.000,E1 336.975} C_DIS
LIN {X -0.047,Y -179.803,Z 1691.849,A 0.000,B 0.000,C 90.000,E1 332.743} C_DIS
LIN {X 0.069,Y -184.434,Z 1691.830,A 0.000,B 0.000,C 90.000,E1 329.331} C_DIS
LIN {X 0.032,Y -188.559,Z 1691.816,A 0.000,B 0.000,C 90.000,E1 326.834} C_DIS
LIN {X -0.022,Y -195.053,Z 1691.797,A 0.000,B 0.000,C 90.000,E1 323.543} C_DIS
LIN {X 0.014,Y -201.616,Z 1691.782,A 0.000,B 0.000,C 90.000,E1 320.678} C_DIS
LIN {X -0.008,Y -209.137,Z 1691.766,A 0.000,B 0.000,C 90.000,E1 317.877} C_DIS
LIN {X -0.024,Y -217.722,Z 1691.751,A 0.000,B 0.000,C 90.000,E1 315.121} C_DIS
LIN {X 0.006,Y -227.422,Z 1691.736,A 0.000,B 0.000,C 90.000,E1 312.405} C_DIS
LIN {X -0.028,Y -236.622,Z 1691.723,A 0.000,B 0.000,C 90.000,E1 310.135} C_DIS
LIN {X 0.033,Y -245.201,Z 1691.713,A 0.000,B 0.000,C 90.000,E1 308.257} C_DIS
LIN {X 0.037,Y -254.624,Z 1691.702,A 0.000,B 0.000,C 90.000,E1 306.423} C_DIS
LIN {X -0.036,Y -271.316,Z 1691.687,A 0.000,B 0.000,C 90.000,E1 303.579} C_DIS
LIN {X 0.034,Y -289.812,Z 1691.671,A 0.000,B 0.000,C 90.000,E1 300.797} C_DIS
LIN {X 0.148,Y -309.419,Z 1691.656,A 0.000,B 0.000,C 90.000,E1 298.103} C_DIS
LIN {X 0.036,Y -324.531,Z 1691.646,A 0.000,B 0.000,C 90.000,E1 296.181} C_DIS
LIN {X 0.067,Y -339.628,Z 1691.635,A 0.000,B 0.000,C 90.000,E1 294.283} C_DIS
LIN {X -0.024,Y -354.952,Z 1691.625,A 0.000,B 0.000,C 90.000,E1 292.461} C_DIS
LIN {X 0.168,Y -364.946,Z 1691.618,A 0.000,B 0.000,C 90.000,E1 291.227} C_DIS
LIN {X 0.015,Y -374.508,Z 1691.611,A 0.000,B 0.000,C 90.000,E1 290.066} C_DIS
LIN {X -0.145,Y -381.123,Z 1691.607,A 0.000,B 0.000,C 90.000,E1 289.214} C_DIS
LIN {X 0.113,Y -387.067,Z 1691.602,A 0.000,B 0.000,C 90.000,E1 288.308} C_DIS
LIN {X -0.089,Y -390.550,Z 1691.599,A 0.000,B 0.000,C 90.000,E1 287.764} C_DIS
LIN {X -0.110,Y -394.961,Z 1691.594,A 0.000,B 0.000,C 90.000,E1 286.913} C_DIS
LIN {X 0.110,Y -397.384,Z 1691.591,A 0.000,B 0.000,C 90.000,E1 286.315} C_DIS
LIN {X 0.033,Y -400.299,Z 1691.586,A 0.000,B 0.000,C 90.000,E1 285.481} C_DIS
LIN {X -0.208,Y -401.817,Z 1691.583,A 0.000,B 0.000,C 90.000,E1 284.954} C_DIS
LIN {X 0.056,Y -402.945,Z 1691.580,A 0.000,B 0.000,C 90.000,E1 284.356} C_DIS
LIN {X -0.163,Y -403.683,Z 1691.577,A 0.000,B 0.000,C 90.000,E1 283.828} C_DIS
LIN {X 0.020,Y -404.048,Z 1691.574,A 0.000,B 0.000,C 90.000,E1 283.244} C_DIS
LIN {X -0.095,Y -403.911,Z 1691.570,A 0.000,B 0.000,C 90.000,E1 282.703} C_DIS
LIN {X 0.094,Y -403.375,Z 1691.567,A 0.000,B 0.000,C 90.000,E1 282.119} C_DIS
LIN {X -0.111,Y -402.388,Z 1691.564,A 0.000,B 0.000,C 90.000,E1 281.591} C_DIS
LIN {X 0.074,Y -400.780,Z 1691.561,A 0.000,B 0.000,C 90.000,E1 281.007} C_DIS
LIN {X -0.213,Y -398.795,Z 1691.558,A 0.000,B 0.000,C 90.000,E1 280.489} C_DIS
LIN {X -0.043,Y -396.180,Z 1691.555,A 0.000,B 0.000,C 90.000,E1 279.905} C_DIS
LIN {X 0.103,Y -393.168,Z 1691.552,A 0.000,B 0.000,C 90.000,E1 279.321} C_DIS
LIN {X -0.162,Y -387.983,Z 1691.547,A 0.000,B 0.000,C 90.000,E1 278.511} C_DIS
LIN {X -0.078,Y -382.252,Z 1691.542,A 0.000,B 0.000,C 90.000,E1 277.644} C_DIS
LIN {X -0.053,Y -375.705,Z 1691.538,A 0.000,B 0.000,C 90.000,E1 276.777} C_DIS
LIN {X -0.080,Y -370.607,Z 1691.534,A 0.000,B 0.000,C 90.000,E1 276.201} C_DIS
LIN {X -0.012,Y -364.978,Z 1691.531,A 0.000,B 0.000,C 90.000,E1 275.625} C_DIS
LIN {X -0.053,Y -359.060,Z 1691.528,A 0.000,B 0.000,C 90.000,E1 275.106} C_DIS
LIN {X 0.156,Y -352.939,Z 1691.526,A 0.000,B 0.000,C 90.000,E1 274.588} C_DIS
LIN {X -0.108,Y -346.484,Z 1691.523,A 0.000,B 0.000,C 90.000,E1 274.188} C_DIS
LIN {X -0.077,Y -339.975,Z 1691.521,A 0.000,B 0.000,C 90.000,E1 273.784} C_DIS
LIN {X -0.158,Y -330.035,Z 1691.518,A 0.000,B 0.000,C 90.000,E1 273.269} C_DIS
LIN {X -0.143,Y -320.019,Z 1691.516,A 0.000,B 0.000,C 90.000,E1 272.808} C_DIS
LIN {X -0.075,Y -313.250,Z 1691.514,A 0.000,B 0.000,C 90.000,E1 272.522} C_DIS
LIN {X -0.131,Y -302.832,Z 1691.512,A 0.000,B 0.000,C 90.000,E1 272.178} C_DIS
LIN {X 0.127,Y -292.763,Z 1691.510,A 0.000,B 0.000,C 90.000,E1 271.835} C_DIS
LIN {X -0.009,Y -281.323,Z 1691.509,A 0.000,B 0.000,C 90.000,E1 271.604} C_DIS
LIN {X -0.121,Y -273.345,Z 1691.508,A 0.000,B 0.000,C 90.000,E1 271.489} C_DIS
LIN {X 0.018,Y -260.111,Z 1691.507,A 0.000,B 0.000,C 90.000,E1 271.318} C_DIS
LIN {X -0.106,Y -251.646,Z 1691.507,A 0.000,B 0.000,C 90.000,E1 271.318} C_DIS
LIN {X 0.110,Y -241.031,Z 1691.507,A 0.000,B 0.000,C 90.000,E1 271.260} C_DIS
LIN {X 0.067,Y -199.858,Z 1691.507,A 0.000,B 0.000,C 90.000,E1 271.260} C_DIS
LIN {X 0.038,Y -183.074,Z 1691.507,A 0.000,B 0.000,C 90.000,E1 271.203} C_DIS
LIN {X 0.018,Y -181.410,Z 1691.507,A 0.000,B 0.000,C 90.000,E1 271.203} C_DIS
LIN {X 0.064,Y -181.581,Z 1691.502,A 0.000,B 0.000,C 90.000,E1 270.286} C_DIS
LIN {X 0.039,Y -180.900,Z 1691.474,A 0.000,B 0.000,C 90.000,E1 265.241} C_DIS
LIN {X -0.011,Y -180.223,Z 1691.464,A 0.000,B 0.000,C 90.000,E1 263.571} C_DIS
LIN {X -0.058,Y -179.038,Z 1691.446,A 0.000,B 0.000,C 90.000,E1 260.208} C_DIS
LIN {X 0.005,Y -178.703,Z 1691.441,A 0.000,B 0.000,C 90.000,E1 259.342} C_DIS
LIN {X -0.055,Y -175.752,Z 1691.412,A 0.000,B 0.000,C 90.000,E1 254.267} C_DIS
LIN {X -0.051,Y -171.936,Z 1691.384,A 0.000,B 0.000,C 90.000,E1 249.135} C_DIS
LIN {X -0.075,Y -171.315,Z 1691.379,A 0.000,B 0.000,C 90.000,E1 248.284} C_DIS
LIN {X -0.022,Y -167.574,Z 1691.355,A 0.000,B 0.000,C 90.000,E1 243.948} C_DIS
LIN {X -0.082,Y -166.206,Z 1691.346,A 0.000,B 0.000,C 90.000,E1 242.231} C_DIS
LIN {X -0.093,Y -162.971,Z 1691.326,A 0.000,B 0.000,C 90.000,E1 238.742} C_DIS
LIN {X -0.046,Y -160.883,Z 1691.312,A 0.000,B 0.000,C 90.000,E1 236.087} C_DIS
LIN {X -0.067,Y -157.654,Z 1691.292,A 0.000,B 0.000,C 90.000,E1 232.557} C_DIS
LIN {X 0.091,Y -155.692,Z 1691.277,A 0.000,B 0.000,C 90.000,E1 229.828} C_DIS
LIN {X -0.073,Y -151.956,Z 1691.252,A 0.000,B 0.000,C 90.000,E1 225.405} C_DIS
LIN {X -0.056,Y -150.197,Z 1691.237,A 0.000,B 0.000,C 90.000,E1 222.690} C_DIS
LIN {X 0.075,Y -146.967,Z 1691.212,A 0.000,B 0.000,C 90.000,E1 218.096} C_DIS
LIN {X -0.022,Y -145.554,Z 1691.197,A 0.000,B 0.000,C 90.000,E1 215.391} C_DIS
LIN {X -0.022,Y -142.947,Z 1691.171,A 0.000,B 0.000,C 90.000,E1 210.797} C_DIS
LIN {X 0.035,Y -141.572,Z 1691.151,A 0.000,B 0.000,C 90.000,E1 207.078} C_DIS
LIN {X -0.043,Y -139.413,Z 1691.114,A 0.000,B 0.000,C 90.000,E1 200.610} C_DIS
LIN {X 0.008,Y -139.136,Z 1691.104,A 0.000,B 0.000,C 90.000,E1 198.725} C_DIS
LIN {X 0.036,Y -138.349,Z 1691.057,A 0.000,B 0.000,C 90.000,E1 190.310} C_DIS
LIN {X 0.024,Y -139.495,Z 1691.005,A 0.000,B 0.000,C 90.000,E1 180.974} C_DIS
LIN {X -0.036,Y -141.110,Z 1690.974,A 0.000,B 0.000,C 90.000,E1 175.412} C_DIS
LIN {X 0.059,Y -142.489,Z 1690.959,A 0.000,B 0.000,C 90.000,E1 172.591} C_DIS
LIN {X 0.006,Y -144.741,Z 1690.933,A 0.000,B 0.000,C 90.000,E1 167.993} C_DIS
LIN {X -0.044,Y -147.348,Z 1690.913,A 0.000,B 0.000,C 90.000,E1 164.338} C_DIS
LIN {X 0.020,Y -150.672,Z 1690.888,A 0.000,B 0.000,C 90.000,E1 159.752} C_DIS
LIN {X -0.099,Y -154.151,Z 1690.867,A 0.000,B 0.000,C 90.000,E1 156.177} C_DIS
LIN {X 0.036,Y -157.581,Z 1690.848,A 0.000,B 0.000,C 90.000,E1 152.538} C_DIS
LIN {X -0.013,Y -161.829,Z 1690.828,A 0.000,B 0.000,C 90.000,E1 148.997} C_DIS
LIN {X 0.006,Y -166.020,Z 1690.808,A 0.000,B 0.000,C 90.000,E1 145.468} C_DIS
LIN {X -0.003,Y -171.021,Z 1690.789,A 0.000,B 0.000,C 90.000,E1 141.984} C_DIS
LIN {X 0.028,Y -175.891,Z 1690.770,A 0.000,B 0.000,C 90.000,E1 138.528} C_DIS
LIN {X -0.096,Y -181.496,Z 1690.751,A 0.000,B 0.000,C 90.000,E1 135.162} C_DIS
LIN {X 0.040,Y -187.012,Z 1690.732,A 0.000,B 0.000,C 90.000,E1 131.757} C_DIS
LIN {X 0.042,Y -190.130,Z 1690.723,A 0.000,B 0.000,C 90.000,E1 130.092} C_DIS
LIN {X 0.061,Y -195.900,Z 1690.704,A 0.000,B 0.000,C 90.000,E1 126.790} C_DIS
LIN {X 0.018,Y -200.731,Z 1690.691,A 0.000,B 0.000,C 90.000,E1 124.358} C_DIS
LIN {X 0.043,Y -206.620,Z 1690.673,A 0.000,B 0.000,C 90.000,E1 121.131} C_DIS
LIN {X -0.001,Y -208.523,Z 1690.668,A 0.000,B 0.000,C 90.000,E1 120.207} C_DIS
LIN {X -0.037,Y -330.485,Z 1690.668,A 0.000,B 0.000,C 90.000,E1 120.207} C_DIS
LIN {X -0.066,Y -333.129,Z 1690.668,A 0.000,B 0.000,C 90.000,E1 120.178} C_DIS
LIN {X 0.067,Y -336.912,Z 1690.667,A 0.000,B 0.000,C 90.000,E1 120.001} C_DIS
LIN {X -0.091,Y -339.134,Z 1690.666,A 0.000,B 0.000,C 90.000,E1 119.873} C_DIS
LIN {X 0.056,Y -342.215,Z 1690.664,A 0.000,B 0.000,C 90.000,E1 119.539} C_DIS
LIN {X -0.063,Y -344.204,Z 1690.663,A 0.000,B 0.000,C 90.000,E1 119.283} C_DIS
LIN {X -0.014,Y -345.763,Z 1690.661,A 0.000,B 0.000,C 90.000,E1 118.999} C_DIS
LIN {X -0.092,Y -359.877,Z 1690.644,A 0.000,B 0.000,C 90.000,E1 115.976} C_DIS
LIN {X 0.210,Y -374.103,Z 1690.629,A 0.000,B 0.000,C 90.000,E1 113.259} C_DIS
LIN {X -0.019,Y -388.115,Z 1690.616,A 0.000,B 0.000,C 90.000,E1 110.972} C_DIS
LIN {X -0.186,Y -403.512,Z 1690.604,A 0.000,B 0.000,C 90.000,E1 108.725} C_DIS
LIN {X -0.103,Y -420.399,Z 1690.592,A 0.000,B 0.000,C 90.000,E1 106.496} C_DIS
LIN {X 0.168,Y -438.894,Z 1690.580,A 0.000,B 0.000,C 90.000,E1 104.300} C_DIS
LIN {X 0.162,Y -458.695,Z 1690.568,A 0.000,B 0.000,C 90.000,E1 102.243} C_DIS
LIN {X 0.018,Y -479.083,Z 1690.558,A 0.000,B 0.000,C 90.000,E1 100.366} C_DIS
LIN {X 0.159,Y -502.623,Z 1690.547,A 0.000,B 0.000,C 90.000,E1 98.398} C_DIS
LIN {X -0.073,Y -504.933,Z 1690.546,A 0.000,B 0.000,C 90.000,E1 98.219} C_DIS
LIN {X 0.121,Y -506.685,Z 1690.544,A 0.000,B 0.000,C 90.000,E1 97.992} C_DIS
LIN {X 0.063,Y -508.263,Z 1690.543,A 0.000,B 0.000,C 90.000,E1 97.757} C_DIS
LIN {X -0.065,Y -509.438,Z 1690.542,A 0.000,B 0.000,C 90.000,E1 97.530} C_DIS
LIN {X -0.233,Y -510.836,Z 1690.539,A 0.000,B 0.000,C 90.000,E1 97.068} C_DIS
LIN {X 0.113,Y -511.166,Z 1690.536,A 0.000,B 0.000,C 90.000,E1 96.549} C_DIS
LIN {X -0.040,Y -510.480,Z 1690.534,A 0.000,B 0.000,C 90.000,E1 96.087} C_DIS
LIN {X -0.193,Y -508.660,Z 1690.531,A 0.000,B 0.000,C 90.000,E1 95.625} C_DIS
LIN {X 0.258,Y -507.214,Z 1690.530,A 0.000,B 0.000,C 90.000,E1 95.334} C_DIS
LIN {X 0.026,Y -494.832,Z 1690.520,A 0.000,B 0.000,C 90.000,E1 93.669} C_DIS
LIN {X 0.184,Y -484.070,Z 1690.512,A 0.000,B 0.000,C 90.000,E1 92.178} C_DIS
LIN {X -0.028,Y -471.418,Z 1690.503,A 0.000,B 0.000,C 90.000,E1 90.458} C_DIS
LIN {X 0.190,Y -460.537,Z 1690.494,A 0.000,B 0.000,C 90.000,E1 88.912} C_DIS
LIN {X 0.222,Y -449.519,Z 1690.485,A 0.000,B 0.000,C 90.000,E1 87.364} C_DIS
LIN {X 0.093,Y -438.273,Z 1690.477,A 0.000,B 0.000,C 90.000,E1 85.812} C_DIS
LIN {X -0.047,Y -424.972,Z 1690.466,A 0.000,B 0.000,C 90.000,E1 83.970} C_DIS
LIN {X 0.197,Y -408.331,Z 1690.453,A 0.000,B 0.000,C 90.000,E1 81.489} C_DIS
LIN {X -0.094,Y -387.366,Z 1690.434,A 0.000,B 0.000,C 90.000,E1 78.173} C_DIS
LIN {X -0.127,Y -374.107,Z 1690.422,A 0.000,B 0.000,C 90.000,E1 75.880} C_DIS
LIN {X 0.065,Y -361.222,Z 1690.408,A 0.000,B 0.000,C 90.000,E1 73.504} C_DIS
LIN {X 0.183,Y -347.154,Z 1690.393,A 0.000,B 0.000,C 90.000,E1 70.786} C_DIS
LIN {X 0.140,Y -332.530,Z 1690.376,A 0.000,B 0.000,C 90.000,E1 67.720} C_DIS
LIN {X -0.041,Y -319.926,Z 1690.361,A 0.000,B 0.000,C 90.000,E1 64.921} C_DIS
LIN {X -0.069,Y -308.992,Z 1690.346,A 0.000,B 0.000,C 90.000,E1 62.359} C_DIS
LIN {X -0.095,Y -299.644,Z 1690.334,A 0.000,B 0.000,C 90.000,E1 60.078} C_DIS
LIN {X -0.035,Y -290.092,Z 1690.321,A 0.000,B 0.000,C 90.000,E1 57.740} C_DIS
LIN {X -0.076,Y -281.780,Z 1690.309,A 0.000,B 0.000,C 90.000,E1 55.722} C_DIS
LIN {X 0.119,Y -273.202,Z 1690.298,A 0.000,B 0.000,C 90.000,E1 53.623} C_DIS
LIN {X -0.149,Y -261.808,Z 1690.282,A 0.000,B 0.000,C 90.000,E1 50.884} C_DIS
LIN {X 0.134,Y -252.093,Z 1690.269,A 0.000,B 0.000,C 90.000,E1 48.324} C_DIS
LIN {X -0.037,Y -240.285,Z 1690.250,A 0.000,B 0.000,C 90.000,E1 45.081} C_DIS
LIN {X -0.001,Y -229.525,Z 1690.232,A 0.000,B 0.000,C 90.000,E1 41.714} C_DIS
LIN {X 0.002,Y -220.818,Z 1690.215,A 0.000,B 0.000,C 90.000,E1 38.669} C_DIS
LIN {X -0.087,Y -212.937,Z 1690.198,A 0.000,B 0.000,C 90.000,E1 35.598} C_DIS
LIN {X 0.033,Y -205.745,Z 1690.180,A 0.000,B 0.000,C 90.000,E1 32.418} C_DIS
LIN {X 0.095,Y -199.212,Z 1690.162,A 0.000,B 0.000,C 90.000,E1 29.205} C_DIS
LIN {X 0.052,Y -193.242,Z 1690.144,A 0.000,B 0.000,C 90.000,E1 25.976} C_DIS
LIN {X -0.032,Y -187.795,Z 1690.126,A 0.000,B 0.000,C 90.000,E1 22.717} C_DIS
LIN {X -0.038,Y -182.955,Z 1690.108,A 0.000,B 0.000,C 90.000,E1 19.396} C_DIS
LIN {X -0.002,Y -178.760,Z 1690.089,A 0.000,B 0.000,C 90.000,E1 16.024} C_DIS
LIN {X 0.025,Y -174.510,Z 1690.065,A 0.000,B 0.000,C 90.000,E1 11.771} C_DIS
LIN {X -0.088,Y -170.754,Z 1690.037,A 0.000,B 0.000,C 90.000,E1 6.663} C_DIS
LIN {X 0.041,Y -168.241,Z 1690.008,A 0.000,B 0.000,C 90.000,E1 1.432} C_DIS
LIN {X -0.083,Y -169.192,Z 1689.920,A 0.000,B 0.000,C 90.000,E1 345.644} C_DIS
LIN {X 0.011,Y -172.168,Z 1689.891,A 0.000,B 0.000,C 90.000,E1 340.423} C_DIS
LIN {X 0.096,Y -175.978,Z 1689.867,A 0.000,B 0.000,C 90.000,E1 336.102} C_DIS
LIN {X -0.053,Y -179.839,Z 1689.849,A 0.000,B 0.000,C 90.000,E1 332.743} C_DIS
LIN {X 0.062,Y -184.514,Z 1689.830,A 0.000,B 0.000,C 90.000,E1 329.331} C_DIS
LIN {X 0.027,Y -188.664,Z 1689.816,A 0.000,B 0.000,C 90.000,E1 326.834} C_DIS
LIN {X -0.024,Y -195.182,Z 1689.797,A 0.000,B 0.000,C 90.000,E1 323.543} C_DIS
LIN {X 0.015,Y -201.757,Z 1689.782,A 0.000,B 0.000,C 90.000,E1 320.678} C_DIS
LIN {X -0.004,Y -209.303,Z 1689.766,A 0.000,B 0.000,C 90.000,E1 317.877} C_DIS
LIN {X -0.016,Y -217.922,Z 1689.751,A 0.000,B 0.000,C 90.000,E1 315.121} C_DIS
LIN {X 0.019,Y -227.625,Z 1689.736,A 0.000,B 0.000,C 90.000,E1 312.405} C_DIS
LIN {X -0.011,Y -236.828,Z 1689.723,A 0.000,B 0.000,C 90.000,E1 310.135} C_DIS
LIN {X 0.054,Y -245.403,Z 1689.713,A 0.000,B 0.000,C 90.000,E1 308.257} C_DIS
LIN {X 0.062,Y -254.824,Z 1689.702,A 0.000,B 0.000,C 90.000,E1 306.423} C_DIS
LIN {X -0.005,Y -271.464,Z 1689.687,A 0.000,B 0.000,C 90.000,E1 303.579} C_DIS
LIN {X 0.071,Y -289.943,Z 1689.671,A 0.000,B 0.000,C 90.000,E1 300.797} C_DIS
LIN {X -0.082,Y -309.516,Z 1689.656,A 0.000,B 0.000,C 90.000,E1 298.153} C_DIS
LIN {X 0.082,Y -324.616,Z 1689.646,A 0.000,B 0.000,C 90.000,E1 296.181} C_DIS
LIN {X -0.192,Y -339.678,Z 1689.635,A 0.000,B 0.000,C 90.000,E1 294.335} C_DIS
LIN {X -0.020,Y -355.064,Z 1689.625,A 0.000,B 0.000,C 90.000,E1 292.461} C_DIS
LIN {X -0.087,Y -367.450,Z 1689.616,A 0.000,B 0.000,C 90.000,E1 290.972} C_DIS
LIN {X 0.031,Y -374.558,Z 1689.611,A 0.000,B 0.000,C 90.000,E1 290.066} C_DIS
LIN {X -0.128,Y -381.155,Z 1689.607,A 0.000,B 0.000,C 90.000,E1 289.214} C_DIS
LIN {X 0.130,Y -387.104,Z 1689.602,A 0.000,B 0.000,C 90.000,E1 288.308} C_DIS
LIN {X -0.072,Y -390.625,Z 1689.599,A 0.000,B 0.000,C 90.000,E1 287.764} C_DIS
LIN {X 0.122,Y -393.680,Z 1689.595,A 0.000,B 0.000,C 90.000,E1 287.166} C_DIS
LIN {X 0.129,Y -397.463,Z 1689.591,A 0.000,B 0.000,C 90.000,E1 286.315} C_DIS
LIN {X 0.052,Y -400.422,Z 1689.586,A 0.000,B 0.000,C 90.000,E1 285.481} C_DIS
LIN {X -0.187,Y -401.936,Z 1689.583,A 0.000,B 0.000,C 90.000,E1 284.954} C_DIS
LIN {X 0.077,Y -403.082,Z 1689.580,A 0.000,B 0.000,C 90.000,E1 284.356} C_DIS
LIN {X -0.141,Y -403.871,Z 1689.577,A 0.000,B 0.000,C 90.000,E1 283.828} C_DIS
LIN {X 0.043,Y -404.203,Z 1689.574,A 0.000,B 0.000,C 90.000,E1 283.244} C_DIS
LIN {X -0.071,Y -404.120,Z 1689.571,A 0.000,B 0.000,C 90.000,E1 282.703} C_DIS
LIN {X 0.119,Y -403.597,Z 1689.567,A 0.000,B 0.000,C 90.000,E1 282.119} C_DIS
LIN {X -0.085,Y -402.591,Z 1689.564,A 0.000,B 0.000,C 90.000,E1 281.591} C_DIS
LIN {X 0.101,Y -400.992,Z 1689.561,A 0.000,B 0.000,C 90.000,E1 281.007} C_DIS
LIN {X -0.185,Y -399.021,Z 1689.558,A 0.000,B 0.000,C 90.000,E1 280.489} C_DIS
LIN {X 0.061,Y -394.966,Z 1689.553,A 0.000,B 0.000,C 90.000,E1 279.613} C_DIS
LIN {X -0.184,Y -389.984,Z 1689.549,A 0.000,B 0.000,C 90.000,E1 278.803} C_DIS
LIN {X -0.087,Y -384.422,Z 1689.544,A 0.000,B 0.000,C 90.000,E1 277.936} C_DIS
LIN {X -0.034,Y -378.175,Z 1689.539,A 0.000,B 0.000,C 90.000,E1 277.068} C_DIS
LIN {X -0.004,Y -373.380,Z 1689.536,A 0.000,B 0.000,C 90.000,E1 276.486} C_DIS
LIN {X -0.045,Y -367.853,Z 1689.533,A 0.000,B 0.000,C 90.000,E1 275.910} C_DIS
LIN {X 0.127,Y -362.021,Z 1689.530,A 0.000,B 0.000,C 90.000,E1 275.334} C_DIS
LIN {X 0.128,Y -355.821,Z 1689.527,A 0.000,B 0.000,C 90.000,E1 274.821} C_DIS
LIN {X 0.102,Y -349.425,Z 1689.524,A 0.000,B 0.000,C 90.000,E1 274.359} C_DIS
LIN {X 0.036,Y -342.848,Z 1689.522,A 0.000,B 0.000,C 90.000,E1 273.955} C_DIS
LIN {X -0.120,Y -336.355,Z 1689.520,A 0.000,B 0.000,C 90.000,E1 273.612} C_DIS
LIN {X 0.046,Y -326.555,Z 1689.517,A 0.000,B 0.000,C 90.000,E1 273.094} C_DIS
LIN {X 0.136,Y -316.447,Z 1689.515,A 0.000,B 0.000,C 90.000,E1 272.636} C_DIS
LIN {X -0.017,Y -306.325,Z 1689.513,A 0.000,B 0.000,C 90.000,E1 272.293} C_DIS
LIN {X 0.130,Y -296.100,Z 1689.511,A 0.000,B 0.000,C 90.000,E1 271.949} C_DIS
LIN {X 0.061,Y -288.938,Z 1689.510,A 0.000,B 0.000,C 90.000,E1 271.776} C_DIS
LIN {X 0.040,Y -277.356,Z 1689.509,A 0.000,B 0.000,C 90.000,E1 271.547} C_DIS
LIN {X -0.034,Y -268.286,Z 1689.508,A 0.000,B 0.000,C 90.000,E1 271.432} C_DIS
LIN {X 0.115,Y -259.284,Z 1689.507,A 0.000,B 0.000,C 90.000,E1 271.318} C_DIS
LIN {X 0.019,Y -249.316,Z 1689.507,A 0.000,B 0.000,C 90.000,E1 271.318} C_DIS
LIN {X -0.010,Y -240.443,Z 1689.507,A 0.000,B 0.000,C 90.000,E1 271.318} C_DIS
LIN {X -0.035,Y -220.226,Z 1689.507,A 0.000,B 0.000,C 90.000,E1 271.318} C_DIS
LIN {X -0.056,Y -206.985,Z 1689.507,A 0.000,B 0.000,C 90.000,E1 271.318} C_DIS
LIN {X -0.057,Y -189.396,Z 1689.507,A 0.000,B 0.000,C 90.000,E1 271.260} C_DIS
LIN {X 0.068,Y -184.097,Z 1689.507,A 0.000,B 0.000,C 90.000,E1 271.203} C_DIS
LIN {X 0.047,Y -181.408,Z 1689.507,A 0.000,B 0.000,C 90.000,E1 271.203} C_DIS
LIN {X -0.057,Y -181.580,Z 1689.502,A 0.000,B 0.000,C 90.000,E1 270.344} C_DIS
LIN {X -0.081,Y -180.902,Z 1689.474,A 0.000,B 0.000,C 90.000,E1 265.298} C_DIS
LIN {X 0.048,Y -180.232,Z 1689.464,A 0.000,B 0.000,C 90.000,E1 263.571} C_DIS
LIN {X 0.064,Y -178.715,Z 1689.441,A 0.000,B 0.000,C 90.000,E1 259.342} C_DIS
LIN {X -0.043,Y -175.763,Z 1689.413,A 0.000,B 0.000,C 90.000,E1 254.283} C_DIS
LIN {X 0.006,Y -171.947,Z 1689.384,A 0.000,B 0.000,C 90.000,E1 249.135} C_DIS
LIN {X -0.017,Y -171.334,Z 1689.379,A 0.000,B 0.000,C 90.000,E1 248.284} C_DIS
LIN {X 0.035,Y -167.589,Z 1689.355,A 0.000,B 0.000,C 90.000,E1 243.948} C_DIS
LIN {X -0.026,Y -166.226,Z 1689.346,A 0.000,B 0.000,C 90.000,E1 242.231} C_DIS
LIN {X -0.037,Y -162.987,Z 1689.326,A 0.000,B 0.000,C 90.000,E1 238.742} C_DIS
LIN {X 0.010,Y -160.904,Z 1689.312,A 0.000,B 0.000,C 90.000,E1 236.087} C_DIS
LIN {X -0.012,Y -157.670,Z 1689.292,A 0.000,B 0.000,C 90.000,E1 232.557} C_DIS
LIN {X -0.074,Y -155.709,Z 1689.277,A 0.000,B 0.000,C 90.000,E1 229.908} C_DIS
LIN {X -0.020,Y -151.971,Z 1689.252,A 0.000,B 0.000,C 90.000,E1 225.405} C_DIS
LIN {X -0.002,Y -150.213,Z 1689.237,A 0.000,B 0.000,C 90.000,E1 222.690} C_DIS
LIN {X -0.079,Y -146.978,Z 1689.212,A 0.000,B 0.000,C 90.000,E1 218.177} C_DIS
LIN {X 0.030,Y -145.564,Z 1689.197,A 0.000,B 0.000,C 90.000,E1 215.391} C_DIS
LIN {X 0.029,Y -142.956,Z 1689.171,A 0.000,B 0.000,C 90.000,E1 210.797} C_DIS
LIN {X -0.040,Y -141.582,Z 1689.151,A 0.000,B 0.000,C 90.000,E1 207.129} C_DIS
LIN {X 0.008,Y -139.416,Z 1689.115,A 0.000,B 0.000,C 90.000,E1 200.610} C_DIS
LIN {X 0.059,Y -139.142,Z 1689.104,A 0.000,B 0.000,C 90.000,E1 198.725} C_DIS
LIN {X -0.049,Y -138.347,Z 1689.057,A 0.000,B 0.000,C 90.000,E1 190.366} C_DIS
LIN {X -0.064,Y -139.491,Z 1689.006,A 0.000,B 0.000,C 90.000,E1 181.031} C_DIS
LIN {X 0.016,Y -141.101,Z 1688.975,A 0.000,B 0.000,C 90.000,E1 175.412} C_DIS
LIN {X -0.031,Y -142.479,Z 1688.959,A 0.000,B 0.000,C 90.000,E1 172.648} C_DIS
LIN {X 0.058,Y -144.728,Z 1688.933,A 0.000,B 0.000,C 90.000,E1 167.993} C_DIS
LIN {X 0.010,Y -147.332,Z 1688.913,A 0.000,B 0.000,C 90.000,E1 164.338} C_DIS
LIN {X 0.075,Y -150.655,Z 1688.888,A 0.000,B 0.000,C 90.000,E1 159.752} C_DIS
LIN {X -0.045,Y -154.133,Z 1688.868,A 0.000,B 0.000,C 90.000,E1 156.177} C_DIS
LIN {X 0.018,Y -157.560,Z 1688.848,A 0.000,B 0.000,C 90.000,E1 152.564} C_DIS
LIN {X 0.043,Y -161.803,Z 1688.828,A 0.000,B 0.000,C 90.000,E1 148.997} C_DIS
LIN {X 0.063,Y -165.994,Z 1688.808,A 0.000,B 0.000,C 90.000,E1 145.468} C_DIS
LIN {X 0.056,Y -170.992,Z 1688.789,A 0.000,B 0.000,C 90.000,E1 141.984} C_DIS
LIN {X -0.029,Y -175.862,Z 1688.770,A 0.000,B 0.000,C 90.000,E1 138.566} C_DIS
LIN {X -0.035,Y -181.467,Z 1688.751,A 0.000,B 0.000,C 90.000,E1 135.162} C_DIS
LIN {X 0.102,Y -186.978,Z 1688.732,A 0.000,B 0.000,C 90.000,E1 131.757} C_DIS
LIN {X 0.103,Y -190.094,Z 1688.723,A 0.000,B 0.000,C 90.000,E1 130.092} C_DIS
LIN {X 0.006,Y -195.866,Z 1688.705,A 0.000,B 0.000,C 90.000,E1 126.824} C_DIS
LIN {X -0.085,Y -200.698,Z 1688.691,A 0.000,B 0.000,C 90.000,E1 124.405} C_DIS
LIN {X 0.108,Y -206.584,Z 1688.673,A 0.000,B 0.000,C 90.000,E1 121.131} C_DIS
LIN {X -0.049,Y -208.447,Z 1688.668,A 0.000,B 0.000,C 90.000,E1 120.256} C_DIS
LIN {X -0.113,Y -330.530,Z 1688.668,A 0.000,B 0.000,C 90.000,E1 120.256} C_DIS
LIN {X -0.129,Y -333.648,Z 1688.668,A 0.000,B 0.000,C 90.000,E1 120.207} C_DIS
LIN {X 0.015,Y -339.183,Z 1688.666,A 0.000,B 0.000,C 90.000,E1 119.873} C_DIS
LIN {X 0.163,Y -342.188,Z 1688.664,A 0.000,B 0.000,C 90.000,E1 119.539} C_DIS
LIN {X 0.015,Y -344.173,Z 1688.663,A 0.000,B 0.000,C 90.000,E1 119.283} C_DIS
LIN {X 0.033,Y -345.726,Z 1688.661,A 0.000,B 0.000,C 90.000,E1 118.999} C_DIS
LIN {X -0.044,Y -359.816,Z 1688.644,A 0.000,B 0.000,C 90.000,E1 115.976} C_DIS
LIN {X -0.234,Y -374.037,Z 1688.629,A 0.000,B 0.000,C 90.000,E1 113.334} C_DIS
LIN {X 0.029,Y -388.045,Z 1688.617,A 0.000,B 0.000,C 90.000,E1 110.972} C_DIS
LIN {X -0.138,Y -403.437,Z 1688.604,A 0.000,B 0.000,C 90.000,E1 108.725} C_DIS
LIN {X -0.055,Y -420.319,Z 1688.592,A 0.000,B 0.000,C 90.000,E1 106.496} C_DIS
LIN {X 0.216,Y -438.809,Z 1688.580,A 0.000,B 0.000,C 90.000,E1 104.300} C_DIS
LIN {X 0.208,Y -458.608,Z 1688.568,A 0.000,B 0.000,C 90.000,E1 102.243} C_DIS
LIN {X 0.060,Y -478.995,Z 1688.558,A 0.000,B 0.000,C 90.000,E1 100.366} C_DIS
LIN {X 0.200,Y -502.533,Z 1688.547,A 0.000,B 0.000,C 90.000,E1 98.398} C_DIS
LIN {X -0.034,Y -504.811,Z 1688.546,A 0.000,B 0.000,C 90.000,E1 98.219} C_DIS
LIN {X 0.160,Y -506.541,Z 1688.545,A 0.000,B 0.000,C 90.000,E1 97.992} C_DIS
LIN {X 0.101,Y -508.099,Z 1688.543,A 0.000,B 0.000,C 90.000,E1 97.757} C_DIS
LIN {X -0.026,Y -509.258,Z 1688.542,A 0.000,B 0.000,C 90.000,E1 97.530} C_DIS
LIN {X -0.194,Y -510.631,Z 1688.539,A 0.000,B 0.000,C 90.000,E1 97.068} C_DIS
LIN {X 0.151,Y -510.939,Z 1688.536,A 0.000,B 0.000,C 90.000,E1 96.549} C_DIS
LIN {X -0.004,Y -510.233,Z 1688.534,A 0.000,B 0.000,C 90.000,E1 96.087} C_DIS
LIN {X -0.158,Y -508.389,Z 1688.531,A 0.000,B 0.000,C 90.000,E1 95.625} C_DIS
LIN {X -0.212,Y -506.924,Z 1688.530,A 0.000,B 0.000,C 90.000,E1 95.391} C_DIS
LIN {X 0.180,Y -496.331,Z 1688.522,A 0.000,B 0.000,C 90.000,E1 93.898} C_DIS
LIN {X -0.129,Y -485.600,Z 1688.514,A 0.000,B 0.000,C 90.000,E1 92.465} C_DIS
LIN {X 0.174,Y -472.974,Z 1688.504,A 0.000,B 0.000,C 90.000,E1 90.688} C_DIS
LIN {X -0.048,Y -462.111,Z 1688.495,A 0.000,B 0.000,C 90.000,E1 89.198} C_DIS
LIN {X 0.019,Y -451.120,Z 1688.487,A 0.000,B 0.000,C 90.000,E1 87.650} C_DIS
LIN {X -0.106,Y -439.879,Z 1688.478,A 0.000,B 0.000,C 90.000,E1 86.102} C_DIS
LIN {X 0.202,Y -426.595,Z 1688.468,A 0.000,B 0.000,C 90.000,E1 84.204} C_DIS
LIN {X 0.070,Y -409.849,Z 1688.454,A 0.000,B 0.000,C 90.000,E1 81.781} C_DIS
LIN {X -0.167,Y -388.720,Z 1688.436,A 0.000,B 0.000,C 90.000,E1 78.465} C_DIS
LIN {X -0.164,Y -375.390,Z 1688.423,A 0.000,B 0.000,C 90.000,E1 76.172} C_DIS
LIN {X 0.065,Y -362.453,Z 1688.410,A 0.000,B 0.000,C 90.000,E1 73.795} C_DIS
LIN {X 0.105,Y -348.301,Z 1688.395,A 0.000,B 0.000,C 90.000,E1 71.094} C_DIS
LIN {X 0.086,Y -332.181,Z 1688.376,A 0.000,B 0.000,C 90.000,E1 67.720} C_DIS
LIN {X -0.101,Y -319.604,Z 1688.361,A 0.000,B 0.000,C 90.000,E1 64.921} C_DIS
LIN {X -0.084,Y -307.333,Z 1688.344,A 0.000,B 0.000,C 90.000,E1 62.025} C_DIS
LIN {X -0.148,Y -297.962,Z 1688.332,A 0.000,B 0.000,C 90.000,E1 59.744} C_DIS
LIN {X 0.037,Y -288.369,Z 1688.319,A 0.000,B 0.000,C 90.000,E1 57.375} C_DIS
LIN {X 0.040,Y -279.977,Z 1688.307,A 0.000,B 0.000,C 90.000,E1 55.341} C_DIS
LIN {X -0.030,Y -271.350,Z 1688.296,A 0.000,B 0.000,C 90.000,E1 53.290} C_DIS
LIN {X 0.127,Y -261.397,Z 1688.282,A 0.000,B 0.000,C 90.000,E1 50.803} C_DIS
LIN {X 0.057,Y -250.370,Z 1688.266,A 0.000,B 0.000,C 90.000,E1 47.957} C_DIS
LIN {X 0.012,Y -238.702,Z 1688.248,A 0.000,B 0.000,C 90.000,E1 44.676} C_DIS
LIN {X -0.002,Y -228.108,Z 1688.229,A 0.000,B 0.000,C 90.000,E1 41.310} C_DIS
LIN {X -0.062,Y -218.562,Z 1688.210,A 0.000,B 0.000,C 90.000,E1 37.890} C_DIS
LIN {X 0.094,Y -210.916,Z 1688.193,A 0.000,B 0.000,C 90.000,E1 34.739} C_DIS
LIN {X 0.041,Y -203.924,Z 1688.176,A 0.000,B 0.000,C 90.000,E1 31.592} C_DIS
LIN {X -0.047,Y -197.547,Z 1688.158,A 0.000,B 0.000,C 90.000,E1 28.409} C_DIS
LIN {X -0.042,Y -191.708,Z 1688.140,A 0.000,B 0.000,C 90.000,E1 25.155} C_DIS
LIN {X 0.012,Y -186.438,Z 1688.121,A 0.000,B 0.000,C 90.000,E1 21.844} C_DIS
LIN {X -0.095,Y -181.746,Z 1688.103,A 0.000,B 0.000,C 90.000,E1 18.544} C_DIS
LIN {X 0.031,Y -177.731,Z 1688.084,A 0.000,B 0.000,C 90.000,E1 15.134} C_DIS
LIN {X -0.012,Y -173.709,Z 1688.061,A 0.000,B 0.000,C 90.000,E1 10.894} C_DIS
LIN {X -0.009,Y -170.152,Z 1688.032,A 0.000,B 0.000,C 90.000,E1 5.739} C_DIS
LIN {X 0.000,Y -167.745,Z 1688.000,A 0.000,B 0.000,C 90.000,E1 360.000} C_DIS
LIN {X 0.054,Y -168.789,Z 1687.925,A 0.000,B 0.000,C 90.000,E1 346.464} C_DIS
LIN {X 0.037,Y -171.557,Z 1687.896,A 0.000,B 0.000,C 90.000,E1 341.275} C_DIS
LIN {X 0.037,Y -175.122,Z 1687.872,A 0.000,B 0.000,C 90.000,E1 336.975} C_DIS
LIN {X -0.059,Y -179.895,Z 1687.849,A 0.000,B 0.000,C 90.000,E1 332.743} C_DIS
LIN {X 0.058,Y -184.605,Z 1687.830,A 0.000,B 0.000,C 90.000,E1 329.331} C_DIS
LIN {X 0.024,Y -188.769,Z 1687.816,A 0.000,B 0.000,C 90.000,E1 326.834} C_DIS
LIN {X 0.007,Y -193.573,Z 1687.802,A 0.000,B 0.000,C 90.000,E1 324.356} C_DIS
LIN {X -0.011,Y -198.955,Z 1687.788,A 0.000,B 0.000,C 90.000,E1 321.904} C_DIS
LIN {X -0.072,Y -206.103,Z 1687.773,A 0.000,B 0.000,C 90.000,E1 319.094} C_DIS
LIN {X -0.004,Y -214.271,Z 1687.757,A 0.000,B 0.000,C 90.000,E1 316.296} C_DIS
LIN {X 0.100,Y -223.506,Z 1687.742,A 0.000,B 0.000,C 90.000,E1 313.542} C_DIS
LIN {X -0.058,Y -233.833,Z 1687.727,A 0.000,B 0.000,C 90.000,E1 310.906} C_DIS
LIN {X -0.080,Y -242.051,Z 1687.717,A 0.000,B 0.000,C 90.000,E1 309.036} C_DIS
LIN {X 0.079,Y -253.037,Z 1687.704,A 0.000,B 0.000,C 90.000,E1 306.790} C_DIS
LIN {X 0.060,Y -267.298,Z 1687.691,A 0.000,B 0.000,C 90.000,E1 304.278} C_DIS
LIN {X -0.159,Y -282.925,Z 1687.677,A 0.000,B 0.000,C 90.000,E1 301.878} C_DIS
LIN {X 0.061,Y -297.247,Z 1687.666,A 0.000,B 0.000,C 90.000,E1 299.795} C_DIS
LIN {X -0.109,Y -314.639,Z 1687.653,A 0.000,B 0.000,C 90.000,E1 297.513} C_DIS
LIN {X -0.077,Y -327.183,Z 1687.644,A 0.000,B 0.000,C 90.000,E1 295.899} C_DIS
LIN {X -0.021,Y -344.821,Z 1687.632,A 0.000,B 0.000,C 90.000,E1 293.695} C_DIS
LIN {X 0.077,Y -357.558,Z 1687.623,A 0.000,B 0.000,C 90.000,E1 292.153} C_DIS
LIN {X -0.037,Y -367.475,Z 1687.616,A 0.000,B 0.000,C 90.000,E1 290.972} C_DIS
LIN {X 0.081,Y -374.567,Z 1687.612,A 0.000,B 0.000,C 90.000,E1 290.066} C_DIS
LIN {X -0.077,Y -381.153,Z 1687.607,A 0.000,B 0.000,C 90.000,E1 289.214} C_DIS
LIN {X -0.186,Y -387.107,Z 1687.602,A 0.000,B 0.000,C 90.000,E1 288.362} C_DIS
LIN {X 0.136,Y -392.241,Z 1687.597,A 0.000,B 0.000,C 90.000,E1 287.457} C_DIS
LIN {X -0.038,Y -395.100,Z 1687.594,A 0.000,B 0.000,C 90.000,E1 286.913} C_DIS
LIN {X 0.184,Y -397.549,Z 1687.591,A 0.000,B 0.000,C 90.000,E1 286.315} C_DIS
LIN {X 0.107,Y -400.514,Z 1687.586,A 0.000,B 0.000,C 90.000,E1 285.481} C_DIS
LIN {X -0.132,Y -402.061,Z 1687.583,A 0.000,B 0.000,C 90.000,E1 284.954} C_DIS
LIN {X 0.133,Y -403.230,Z 1687.580,A 0.000,B 0.000,C 90.000,E1 284.356} C_DIS
LIN {X -0.083,Y -404.004,Z 1687.577,A 0.000,B 0.000,C 90.000,E1 283.828} C_DIS
LIN {X 0.101,Y -404.349,Z 1687.574,A 0.000,B 0.000,C 90.000,E1 283.244} C_DIS
LIN {X -0.013,Y -404.303,Z 1687.571,A 0.000,B 0.000,C 90.000,E1 282.703} C_DIS
LIN {X 0.179,Y -403.791,Z 1687.568,A 0.000,B 0.000,C 90.000,E1 282.119} C_DIS
LIN {X -0.024,Y -402.777,Z 1687.564,A 0.000,B 0.000,C 90.000,E1 281.591} C_DIS
LIN {X 0.164,Y -401.252,Z 1687.561,A 0.000,B 0.000,C 90.000,E1 281.007} C_DIS
LIN {X -0.122,Y -399.242,Z 1687.558,A 0.000,B 0.000,C 90.000,E1 280.489} C_DIS
LIN {X 0.050,Y -396.686,Z 1687.555,A 0.000,B 0.000,C 90.000,E1 279.905} C_DIS
LIN {X -0.123,Y -392.000,Z 1687.550,A 0.000,B 0.000,C 90.000,E1 279.086} C_DIS
LIN {X -0.009,Y -386.600,Z 1687.546,A 0.000,B 0.000,C 90.000,E1 278.219} C_DIS
LIN {X 0.053,Y -380.568,Z 1687.541,A 0.000,B 0.000,C 90.000,E1 277.352} C_DIS
LIN {X 0.050,Y -376.012,Z 1687.538,A 0.000,B 0.000,C 90.000,E1 276.777} C_DIS
LIN {X 0.024,Y -370.765,Z 1687.534,A 0.000,B 0.000,C 90.000,E1 276.201} C_DIS
LIN {X 0.080,Y -365.081,Z 1687.531,A 0.000,B 0.000,C 90.000,E1 275.625} C_DIS
LIN {X 0.032,Y -359.066,Z 1687.528,A 0.000,B 0.000,C 90.000,E1 275.106} C_DIS
LIN {X -0.087,Y -352.805,Z 1687.526,A 0.000,B 0.000,C 90.000,E1 274.645} C_DIS
LIN {X 0.023,Y -346.336,Z 1687.523,A 0.000,B 0.000,C 90.000,E1 274.188} C_DIS
LIN {X 0.052,Y -336.474,Z 1687.520,A 0.000,B 0.000,C 90.000,E1 273.612} C_DIS
LIN {X -0.136,Y -326.559,Z 1687.517,A 0.000,B 0.000,C 90.000,E1 273.151} C_DIS
LIN {X -0.012,Y -316.530,Z 1687.515,A 0.000,B 0.000,C 90.000,E1 272.694} C_DIS
LIN {X 0.130,Y -306.405,Z 1687.513,A 0.000,B 0.000,C 90.000,E1 272.293} C_DIS
LIN {X -0.053,Y -296.055,Z 1687.511,A 0.000,B 0.000,C 90.000,E1 272.007} C_DIS
LIN {X 0.062,Y -285.268,Z 1687.510,A 0.000,B 0.000,C 90.000,E1 271.718} C_DIS
LIN {X 0.098,Y -272.889,Z 1687.508,A 0.000,B 0.000,C 90.000,E1 271.489} C_DIS
LIN {X -0.024,Y -258.805,Z 1687.508,A 0.000,B 0.000,C 90.000,E1 271.375} C_DIS
LIN {X -0.070,Y -254.401,Z 1687.508,A 0.000,B 0.000,C 90.000,E1 271.375} C_DIS
LIN {X -0.112,Y -242.943,Z 1687.507,A 0.000,B 0.000,C 90.000,E1 271.375} C_DIS
LIN {X 0.102,Y -238.561,Z 1687.507,A 0.000,B 0.000,C 90.000,E1 271.318} C_DIS
LIN {X 0.069,Y -222.350,Z 1687.507,A 0.000,B 0.000,C 90.000,E1 271.318} C_DIS
LIN {X 0.043,Y -220.032,Z 1687.507,A 0.000,B 0.000,C 90.000,E1 271.318} C_DIS
LIN {X 0.017,Y -211.058,Z 1687.507,A 0.000,B 0.000,C 90.000,E1 271.318} C_DIS
LIN {X 0.008,Y -191.414,Z 1687.507,A 0.000,B 0.000,C 90.000,E1 271.260} C_DIS
LIN {X 0.083,Y -183.216,Z 1687.507,A 0.000,B 0.000,C 90.000,E1 271.203} C_DIS
LIN {X 0.053,Y -181.408,Z 1687.507,A 0.000,B 0.000,C 90.000,E1 271.203} C_DIS
LIN {X 0.084,Y -181.581,Z 1687.502,A 0.000,B 0.000,C 90.000,E1 270.286} C_DIS
LIN {X 0.058,Y -180.901,Z 1687.474,A 0.000,B 0.000,C 90.000,E1 265.241} C_DIS
LIN {X 0.009,Y -180.226,Z 1687.464,A 0.000,B 0.000,C 90.000,E1 263.571} C_DIS
LIN {X -0.038,Y -179.040,Z 1687.446,A 0.000,B 0.000,C 90.000,E1 260.208} C_DIS
LIN {X 0.024,Y -178.707,Z 1687.441,A 0.000,B 0.000,C 90.000,E1 259.342} C_DIS
LIN {X -0.035,Y -175.756,Z 1687.412,A 0.000,B 0.000,C 90.000,E1 254.267} C_DIS
LIN {X -0.033,Y -171.940,Z 1687.384,A 0.000,B 0.000,C 90.000,E1 249.135} C_DIS
LIN {X -0.056,Y -171.322,Z 1687.379,A 0.000,B 0.000,C 90.000,E1 248.284} C_DIS
LIN {X -0.003,Y -167.579,Z 1687.355,A 0.000,B 0.000,C 90.000,E1 243.948} C_DIS
LIN {X -0.064,Y -166.212,Z 1687.346,A 0.000,B 0.000,C 90.000,E1 242.231} C_DIS
LIN {X -0.075,Y -162.977,Z 1687.326,A 0.000,B 0.000,C 90.000,E1 238.742} C_DIS
LIN {X -0.028,Y -160.890,Z 1687.312,A 0.000,B 0.000,C 90.000,E1 236.087} C_DIS
LIN {X -0.049,Y -157.659,Z 1687.292,A 0.000,B 0.000,C 90.000,E1 232.557} C_DIS
LIN {X 0.008,Y -155.697,Z 1687.277,A 0.000,B 0.000,C 90.000,E1 229.865} C_DIS
LIN {X -0.056,Y -151.961,Z 1687.252,A 0.000,B 0.000,C 90.000,E1 225.405} C_DIS
LIN {X -0.039,Y -150.202,Z 1687.237,A 0.000,B 0.000,C 90.000,E1 222.690} C_DIS
LIN {X 0.091,Y -146.970,Z 1687.212,A 0.000,B 0.000,C 90.000,E1 218.096} C_DIS
LIN {X -0.005,Y -145.557,Z 1687.197,A 0.000,B 0.000,C 90.000,E1 215.391} C_DIS
LIN {X -0.005,Y -142.950,Z 1687.171,A 0.000,B 0.000,C 90.000,E1 210.797} C_DIS
LIN {X -0.075,Y -141.576,Z 1687.151,A 0.000,B 0.000,C 90.000,E1 207.129} C_DIS
LIN {X -0.027,Y -139.414,Z 1687.114,A 0.000,B 0.000,C 90.000,E1 200.610} C_DIS
LIN {X 0.026,Y -139.138,Z 1687.104,A 0.000,B 0.000,C 90.000,E1 198.725} C_DIS
LIN {X 0.052,Y -138.348,Z 1687.057,A 0.000,B 0.000,C 90.000,E1 190.310} C_DIS
LIN {X 0.040,Y -139.493,Z 1687.005,A 0.000,B 0.000,C 90.000,E1 180.974} C_DIS
LIN {X -0.019,Y -141.107,Z 1686.974,A 0.000,B 0.000,C 90.000,E1 175.412} C_DIS
LIN {X -0.065,Y -142.486,Z 1686.959,A 0.000,B 0.000,C 90.000,E1 172.648} C_DIS
LIN {X 0.023,Y -144.737,Z 1686.933,A 0.000,B 0.000,C 90.000,E1 167.993} C_DIS
LIN {X -0.027,Y -147.342,Z 1686.913,A 0.000,B 0.000,C 90.000,E1 164.338} C_DIS
LIN {X 0.037,Y -150.666,Z 1686.888,A 0.000,B 0.000,C 90.000,E1 159.752} C_DIS
LIN {X -0.081,Y -154.145,Z 1686.867,A 0.000,B 0.000,C 90.000,E1 156.177} C_DIS
LIN {X 0.054,Y -157.575,Z 1686.848,A 0.000,B 0.000,C 90.000,E1 152.538} C_DIS
LIN {X 0.005,Y -161.820,Z 1686.828,A 0.000,B 0.000,C 90.000,E1 148.997} C_DIS
LIN {X 0.024,Y -166.011,Z 1686.808,A 0.000,B 0.000,C 90.000,E1 145.468} C_DIS
LIN {X 0.016,Y -171.011,Z 1686.789,A 0.000,B 0.000,C 90.000,E1 141.984} C_DIS
LIN {X 0.048,Y -175.882,Z 1686.770,A 0.000,B 0.000,C 90.000,E1 138.528} C_DIS
LIN {X -0.076,Y -181.486,Z 1686.751,A 0.000,B 0.000,C 90.000,E1 135.162} C_DIS
LIN {X 0.060,Y -187.001,Z 1686.732,A 0.000,B 0.000,C 90.000,E1 131.757} C_DIS
LIN {X 0.062,Y -190.118,Z 1686.723,A 0.000,B 0.000,C 90.000,E1 130.092} C_DIS
LIN {X 0.081,Y -195.889,Z 1686.704,A 0.000,B 0.000,C 90.000,E1 126.790} C_DIS
LIN {X -0.128,Y -200.720,Z 1686.691,A 0.000,B 0.000,C 90.000,E1 124.405} C_DIS
LIN {X 0.064,Y -206.608,Z 1686.673,A 0.000,B 0.000,C 90.000,E1 121.131} C_DIS
LIN {X 0.077,Y -208.375,Z 1686.668,A 0.000,B 0.000,C 90.000,E1 120.256} C_DIS
LIN {X 0.087,Y -330.716,Z 1686.668,A 0.000,B 0.000,C 90.000,E1 120.256} C_DIS
LIN {X 0.139,Y -333.143,Z 1686.668,A 0.000,B 0.000,C 90.000,E1 120.207} C_DIS
LIN {X -0.102,Y -336.955,Z 1686.667,A 0.000,B 0.000,C 90.000,E1 120.079} C_DIS
LIN {X 0.116,Y -339.235,Z 1686.666,A 0.000,B 0.000,C 90.000,E1 119.873} C_DIS
LIN {X 0.091,Y -342.393,Z 1686.664,A 0.000,B 0.000,C 90.000,E1 119.539} C_DIS
LIN {X -0.107,Y -344.340,Z 1686.663,A 0.000,B 0.000,C 90.000,E1 119.283} C_DIS
LIN {X 0.163,Y -345.859,Z 1686.661,A 0.000,B 0.000,C 90.000,E1 118.949} C_DIS
LIN {X 0.059,Y -358.446,Z 1686.646,A 0.000,B 0.000,C 90.000,E1 116.232} C_DIS
LIN {X -0.020,Y -372.512,Z 1686.631,A 0.000,B 0.000,C 90.000,E1 113.567} C_DIS
LIN {X 0.062,Y -386.370,Z 1686.618,A 0.000,B 0.000,C 90.000,E1 111.227} C_DIS
LIN {X -0.007,Y -401.600,Z 1686.605,A 0.000,B 0.000,C 90.000,E1 108.960} C_DIS
LIN {X 0.030,Y -418.308,Z 1686.593,A 0.000,B 0.000,C 90.000,E1 106.732} C_DIS
LIN {X -0.171,Y -436.610,Z 1686.581,A 0.000,B 0.000,C 90.000,E1 104.592} C_DIS
LIN {X 0.103,Y -456.322,Z 1686.569,A 0.000,B 0.000,C 90.000,E1 102.479} C_DIS
LIN {X -0.195,Y -476.649,Z 1686.559,A 0.000,B 0.000,C 90.000,E1 100.602} C_DIS
LIN {X -0.130,Y -500.101,Z 1686.548,A 0.000,B 0.000,C 90.000,E1 98.624} C_DIS
LIN {X 0.024,Y -502.750,Z 1686.547,A 0.000,B 0.000,C 90.000,E1 98.398} C_DIS
LIN {X -0.064,Y -506.614,Z 1686.544,A 0.000,B 0.000,C 90.000,E1 97.992} C_DIS
LIN {X -0.130,Y -508.102,Z 1686.543,A 0.000,B 0.000,C 90.000,E1 97.757} C_DIS
LIN {X -0.263,Y -509.205,Z 1686.542,A 0.000,B 0.000,C 90.000,E1 97.530} C_DIS
LIN {X 0.136,Y -510.481,Z 1686.539,A 0.000,B 0.000,C 90.000,E1 97.004} C_DIS
LIN {X -0.088,Y -510.705,Z 1686.536,A 0.000,B 0.000,C 90.000,E1 96.549} C_DIS
LIN {X -0.243,Y -509.908,Z 1686.534,A 0.000,B 0.000,C 90.000,E1 96.087} C_DIS
LIN {X 0.109,Y -507.954,Z 1686.531,A 0.000,B 0.000,C 90.000,E1 95.568} C_DIS
LIN {X -0.052,Y -504.653,Z 1686.528,A 0.000,B 0.000,C 90.000,E1 95.106} C_DIS
LIN {X -0.189,Y -494.029,Z 1686.520,A 0.000,B 0.000,C 90.000,E1 93.669} C_DIS
LIN {X -0.199,Y -481.505,Z 1686.511,A 0.000,B 0.000,C 90.000,E1 91.949} C_DIS
LIN {X 0.025,Y -468.882,Z 1686.501,A 0.000,B 0.000,C 90.000,E1 90.172} C_DIS
LIN {X 0.196,Y -457.969,Z 1686.493,A 0.000,B 0.000,C 90.000,E1 88.625} C_DIS
LIN {X 0.183,Y -446.881,Z 1686.484,A 0.000,B 0.000,C 90.000,E1 87.078} C_DIS
LIN {X 0.007,Y -435.564,Z 1686.475,A 0.000,B 0.000,C 90.000,E1 85.527} C_DIS
LIN {X -0.195,Y -422.265,Z 1686.465,A 0.000,B 0.000,C 90.000,E1 83.685} C_DIS
LIN {X 0.039,Y -405.673,Z 1686.451,A 0.000,B 0.000,C 90.000,E1 81.197} C_DIS
LIN {X 0.045,Y -384.817,Z 1686.432,A 0.000,B 0.000,C 90.000,E1 77.825} C_DIS
LIN {X 0.030,Y -369.920,Z 1686.418,A 0.000,B 0.000,C 90.000,E1 75.227} C_DIS
LIN {X 0.116,Y -357.102,Z 1686.405,A 0.000,B 0.000,C 90.000,E1 72.851} C_DIS
LIN {X 0.139,Y -338.794,Z 1686.385,A 0.000,B 0.000,C 90.000,E1 69.209} C_DIS
LIN {X 0.034,Y -327.400,Z 1686.371,A 0.000,B 0.000,C 90.000,E1 66.741} C_DIS
LIN {X -0.022,Y -317.707,Z 1686.359,A 0.000,B 0.000,C 90.000,E1 64.537} C_DIS
LIN {X -0.062,Y -305.511,Z 1686.342,A 0.000,B 0.000,C 90.000,E1 61.641} C_DIS
LIN {X -0.015,Y -296.121,Z 1686.330,A 0.000,B 0.000,C 90.000,E1 59.331} C_DIS
LIN {X -0.014,Y -287.850,Z 1686.318,A 0.000,B 0.000,C 90.000,E1 57.327} C_DIS
LIN {X -0.095,Y -279.393,Z 1686.307,A 0.000,B 0.000,C 90.000,E1 55.308} C_DIS
LIN {X 0.053,Y -270.763,Z 1686.296,A 0.000,B 0.000,C 90.000,E1 53.210} C_DIS
LIN {X -0.112,Y -259.432,Z 1686.280,A 0.000,B 0.000,C 90.000,E1 50.436} C_DIS
LIN {X -0.055,Y -248.466,Z 1686.264,A 0.000,B 0.000,C 90.000,E1 47.553} C_DIS
LIN {X -0.148,Y -237.000,Z 1686.246,A 0.000,B 0.000,C 90.000,E1 44.271} C_DIS
LIN {X -0.028,Y -226.608,Z 1686.227,A 0.000,B 0.000,C 90.000,E1 40.862} C_DIS
LIN {X -0.054,Y -218.228,Z 1686.210,A 0.000,B 0.000,C 90.000,E1 37.810} C_DIS
LIN {X -0.028,Y -210.624,Z 1686.193,A 0.000,B 0.000,C 90.000,E1 34.692} C_DIS
LIN {X -0.079,Y -203.683,Z 1686.175,A 0.000,B 0.000,C 90.000,E1 31.544} C_DIS
LIN {X 0.011,Y -197.318,Z 1686.157,A 0.000,B 0.000,C 90.000,E1 28.309} C_DIS
LIN {X -0.073,Y -191.508,Z 1686.139,A 0.000,B 0.000,C 90.000,E1 25.079} C_DIS
LIN {X -0.028,Y -186.242,Z 1686.121,A 0.000,B 0.000,C 90.000,E1 21.770} C_DIS
LIN {X 0.027,Y -181.575,Z 1686.102,A 0.000,B 0.000,C 90.000,E1 18.417} C_DIS
LIN {X -0.030,Y -177.569,Z 1686.084,A 0.000,B 0.000,C 90.000,E1 15.064} C_DIS
LIN {X 0.052,Y -173.580,Z 1686.060,A 0.000,B 0.000,C 90.000,E1 10.782} C_DIS
LIN {X 0.053,Y -170.042,Z 1686.031,A 0.000,B 0.000,C 90.000,E1 5.625} C_DIS
LIN {X -0.030,Y -167.589,Z 1685.997,A 0.000,B 0.000,C 90.000,E1 359.542} C_DIS
LIN {X 0.050,Y -168.764,Z 1685.925,A 0.000,B 0.000,C 90.000,E1 346.464} C_DIS
LIN {X 0.033,Y -171.542,Z 1685.896,A 0.000,B 0.000,C 90.000,E1 341.275} C_DIS
LIN {X 0.033,Y -175.147,Z 1685.872,A 0.000,B 0.000,C 90.000,E1 336.975} C_DIS
LIN {X -0.063,Y -179.955,Z 1685.849,A 0.000,B 0.000,C 90.000,E1 332.743} C_DIS
LIN {X 0.056,Y -184.692,Z 1685.830,A 0.000,B 0.000,C 90.000,E1 329.331} C_DIS
LIN {X 0.023,Y -188.875,Z 1685.816,A 0.000,B 0.000,C 90.000,E1 326.834} C_DIS
LIN {X 0.008,Y -193.684,Z 1685.802,A 0.000,B 0.000,C 90.000,E1 324.356} C_DIS
LIN {X -0.008,Y -199.087,Z 1685.788,A 0.000,B 0.000,C 90.000,E1 321.904} C_DIS
LIN {X -0.066,Y -206.254,Z 1685.773,A 0.000,B 0.000,C 90.000,E1 319.094} C_DIS
LIN {X 0.006,Y -214.453,Z 1685.757,A 0.000,B 0.000,C 90.000,E1 316.296} C_DIS
LIN {X 0.114,Y -223.707,Z 1685.742,A 0.000,B 0.000,C 90.000,E1 313.542} C_DIS
LIN {X -0.039,Y -234.029,Z 1685.727,A 0.000,B 0.000,C 90.000,E1 310.906} C_DIS
LIN {X -0.078,Y -244.020,Z 1685.715,A 0.000,B 0.000,C 90.000,E1 308.669} C_DIS
LIN {X 0.108,Y -253.212,Z 1685.704,A 0.000,B 0.000,C 90.000,E1 306.790} C_DIS
LIN {X -0.127,Y -267.459,Z 1685.691,A 0.000,B 0.000,C 90.000,E1 304.326} C_DIS
LIN {X -0.119,Y -283.038,Z 1685.677,A 0.000,B 0.000,C 90.000,E1 301.878} C_DIS
LIN {X 0.098,Y -299.802,Z 1685.664,A 0.000,B 0.000,C 90.000,E1 299.461} C_DIS
LIN {X -0.007,Y -317.266,Z 1685.651,A 0.000,B 0.000,C 90.000,E1 297.180} C_DIS
LIN {X -0.083,Y -329.785,Z 1685.642,A 0.000,B 0.000,C 90.000,E1 295.591} C_DIS
LIN {X 0.042,Y -347.412,Z 1685.630,A 0.000,B 0.000,C 90.000,E1 293.387} C_DIS
LIN {X -0.134,Y -360.041,Z 1685.622,A 0.000,B 0.000,C 90.000,E1 291.897} C_DIS
LIN {X 0.119,Y -369.855,Z 1685.615,A 0.000,B 0.000,C 90.000,E1 290.663} C_DIS
LIN {X -0.083,Y -376.776,Z 1685.610,A 0.000,B 0.000,C 90.000,E1 289.812} C_DIS
LIN {X 0.128,Y -383.209,Z 1685.605,A 0.000,B 0.000,C 90.000,E1 288.906} C_DIS
LIN {X 0.046,Y -388.903,Z 1685.600,A 0.000,B 0.000,C 90.000,E1 288.055} C_DIS
LIN {X -0.149,Y -392.240,Z 1685.597,A 0.000,B 0.000,C 90.000,E1 287.511} C_DIS
LIN {X 0.051,Y -395.132,Z 1685.594,A 0.000,B 0.000,C 90.000,E1 286.913} C_DIS
LIN {X -0.107,Y -397.613,Z 1685.591,A 0.000,B 0.000,C 90.000,E1 286.370} C_DIS
LIN {X 0.200,Y -400.583,Z 1685.586,A 0.000,B 0.000,C 90.000,E1 285.481} C_DIS
LIN {X -0.039,Y -402.166,Z 1685.583,A 0.000,B 0.000,C 90.000,E1 284.954} C_DIS
LIN {X 0.227,Y -403.369,Z 1685.580,A 0.000,B 0.000,C 90.000,E1 284.356} C_DIS
LIN {X 0.011,Y -404.161,Z 1685.577,A 0.000,B 0.000,C 90.000,E1 283.828} C_DIS
LIN {X -0.198,Y -404.557,Z 1685.574,A 0.000,B 0.000,C 90.000,E1 283.300} C_DIS
LIN {X -0.005,Y -404.506,Z 1685.571,A 0.000,B 0.000,C 90.000,E1 282.715} C_DIS
LIN {X -0.119,Y -404.003,Z 1685.568,A 0.000,B 0.000,C 90.000,E1 282.175} C_DIS
LIN {X 0.074,Y -403.007,Z 1685.564,A 0.000,B 0.000,C 90.000,E1 281.591} C_DIS
LIN {X -0.209,Y -401.504,Z 1685.561,A 0.000,B 0.000,C 90.000,E1 281.074} C_DIS
LIN {X -0.023,Y -399.499,Z 1685.558,A 0.000,B 0.000,C 90.000,E1 280.489} C_DIS
LIN {X 0.151,Y -396.956,Z 1685.555,A 0.000,B 0.000,C 90.000,E1 279.905} C_DIS
LIN {X -0.084,Y -392.296,Z 1685.550,A 0.000,B 0.000,C 90.000,E1 279.095} C_DIS
LIN {X 0.094,Y -386.840,Z 1685.546,A 0.000,B 0.000,C 90.000,E1 278.219} C_DIS
LIN {X 0.156,Y -380.783,Z 1685.541,A 0.000,B 0.000,C 90.000,E1 277.352} C_DIS
LIN {X 0.154,Y -376.181,Z 1685.538,A 0.000,B 0.000,C 90.000,E1 276.777} C_DIS
LIN {X 0.127,Y -370.941,Z 1685.535,A 0.000,B 0.000,C 90.000,E1 276.201} C_DIS
LIN {X -0.158,Y -365.207,Z 1685.531,A 0.000,B 0.000,C 90.000,E1 275.682} C_DIS
LIN {X 0.177,Y -359.242,Z 1685.529,A 0.000,B 0.000,C 90.000,E1 275.106} C_DIS
LIN {X 0.072,Y -352.996,Z 1685.526,A 0.000,B 0.000,C 90.000,E1 274.645} C_DIS
LIN {X -0.133,Y -346.575,Z 1685.523,A 0.000,B 0.000,C 90.000,E1 274.245} C_DIS
LIN {X -0.057,Y -336.750,Z 1685.520,A 0.000,B 0.000,C 90.000,E1 273.669} C_DIS
LIN {X 0.098,Y -326.940,Z 1685.518,A 0.000,B 0.000,C 90.000,E1 273.154} C_DIS
LIN {X -0.101,Y -316.877,Z 1685.515,A 0.000,B 0.000,C 90.000,E1 272.751} C_DIS
LIN {X 0.063,Y -307.023,Z 1685.513,A 0.000,B 0.000,C 90.000,E1 272.350} C_DIS
LIN {X -0.137,Y -296.717,Z 1685.511,A 0.000,B 0.000,C 90.000,E1 272.064} C_DIS
LIN {X -0.022,Y -286.082,Z 1685.510,A 0.000,B 0.000,C 90.000,E1 271.776} C_DIS
LIN {X 0.002,Y -273.705,Z 1685.509,A 0.000,B 0.000,C 90.000,E1 271.547} C_DIS
LIN {X -0.037,Y -263.306,Z 1685.508,A 0.000,B 0.000,C 90.000,E1 271.432} C_DIS
LIN {X 0.064,Y -255.254,Z 1685.508,A 0.000,B 0.000,C 90.000,E1 271.375} C_DIS
LIN {X 0.037,Y -246.800,Z 1685.508,A 0.000,B 0.000,C 90.000,E1 271.375} C_DIS
LIN {X -0.043,Y -236.975,Z 1685.508,A 0.000,B 0.000,C 90.000,E1 271.375} C_DIS
LIN {X -0.067,Y -223.961,Z 1685.508,A 0.000,B 0.000,C 90.000,E1 271.375} C_DIS
LIN {X -0.060,Y -196.760,Z 1685.507,A 0.000,B 0.000,C 90.000,E1 271.318} C_DIS
LIN {X -0.074,Y -183.261,Z 1685.507,A 0.000,B 0.000,C 90.000,E1 271.260} C_DIS
LIN {X 0.088,Y -181.406,Z 1685.507,A 0.000,B 0.000,C 90.000,E1 271.203} C_DIS
LIN {X -0.035,Y -181.580,Z 1685.502,A 0.000,B 0.000,C 90.000,E1 270.344} C_DIS
LIN {X -0.060,Y -180.903,Z 1685.474,A 0.000,B 0.000,C 90.000,E1 265.298} C_DIS
LIN {X 0.070,Y -180.235,Z 1685.464,A 0.000,B 0.000,C 90.000,E1 263.571} C_DIS
LIN {X -0.091,Y -178.720,Z 1685.441,A 0.000,B 0.000,C 90.000,E1 259.398} C_DIS
LIN {X -0.022,Y -175.768,Z 1685.413,A 0.000,B 0.000,C 90.000,E1 254.283} C_DIS
LIN {X 0.027,Y -171.951,Z 1685.384,A 0.000,B 0.000,C 90.000,E1 249.135} C_DIS
LIN {X 0.003,Y -171.340,Z 1685.379,A 0.000,B 0.000,C 90.000,E1 248.284} C_DIS
LIN {X -0.018,Y -167.593,Z 1685.355,A 0.000,B 0.000,C 90.000,E1 243.973} C_DIS
LIN {X -0.006,Y -166.233,Z 1685.346,A 0.000,B 0.000,C 90.000,E1 242.231} C_DIS
LIN {X -0.018,Y -162.993,Z 1685.326,A 0.000,B 0.000,C 90.000,E1 238.742} C_DIS
LIN {X 0.030,Y -160.911,Z 1685.312,A 0.000,B 0.000,C 90.000,E1 236.087} C_DIS
LIN {X 0.008,Y -157.676,Z 1685.292,A 0.000,B 0.000,C 90.000,E1 232.557} C_DIS
LIN {X -0.055,Y -155.715,Z 1685.277,A 0.000,B 0.000,C 90.000,E1 229.908} C_DIS
LIN {X 0.000,Y -151.975,Z 1685.252,A 0.000,B 0.000,C 90.000,E1 225.405} C_DIS
LIN {X 0.016,Y -150.219,Z 1685.237,A 0.000,B 0.000,C 90.000,E1 222.690} C_DIS
LIN {X -0.060,Y -146.983,Z 1685.212,A 0.000,B 0.000,C 90.000,E1 218.177} C_DIS
LIN {X 0.049,Y -145.569,Z 1685.197,A 0.000,B 0.000,C 90.000,E1 215.391} C_DIS
LIN {X 0.048,Y -142.960,Z 1685.171,A 0.000,B 0.000,C 90.000,E1 210.797} C_DIS
LIN {X -0.021,Y -141.586,Z 1685.151,A 0.000,B 0.000,C 90.000,E1 207.129} C_DIS
LIN {X 0.026,Y -139.418,Z 1685.115,A 0.000,B 0.000,C 90.000,E1 200.610} C_DIS
LIN {X -0.054,Y -139.144,Z 1685.104,A 0.000,B 0.000,C 90.000,E1 198.779} C_DIS
LIN {X -0.032,Y -138.347,Z 1685.057,A 0.000,B 0.000,C 90.000,E1 190.366} C_DIS
LIN {X -0.046,Y -139.490,Z 1685.006,A 0.000,B 0.000,C 90.000,E1 181.031} C_DIS
LIN {X 0.035,Y -141.097,Z 1684.975,A 0.000,B 0.000,C 90.000,E1 175.412} C_DIS
LIN {X -0.012,Y -142.476,Z 1684.959,A 0.000,B 0.000,C 90.000,E1 172.648} C_DIS
LIN {X 0.077,Y -144.724,Z 1684.933,A 0.000,B 0.000,C 90.000,E1 167.993} C_DIS
LIN {X 0.028,Y -147.326,Z 1684.913,A 0.000,B 0.000,C 90.000,E1 164.338} C_DIS
LIN {X -0.048,Y -150.648,Z 1684.888,A 0.000,B 0.000,C 90.000,E1 159.806} C_DIS
LIN {X -0.025,Y -154.126,Z 1684.868,A 0.000,B 0.000,C 90.000,E1 156.177} C_DIS
LIN {X 0.038,Y -157.553,Z 1684.848,A 0.000,B 0.000,C 90.000,E1 152.564} C_DIS
LIN {X 0.063,Y -161.793,Z 1684.828,A 0.000,B 0.000,C 90.000,E1 148.997} C_DIS
LIN {X -0.054,Y -165.985,Z 1684.808,A 0.000,B 0.000,C 90.000,E1 145.515} C_DIS
LIN {X 0.076,Y -170.982,Z 1684.789,A 0.000,B 0.000,C 90.000,E1 141.984} C_DIS
LIN {X -0.008,Y -175.851,Z 1684.770,A 0.000,B 0.000,C 90.000,E1 138.566} C_DIS
LIN {X -0.013,Y -181.456,Z 1684.751,A 0.000,B 0.000,C 90.000,E1 135.162} C_DIS
LIN {X 0.124,Y -186.966,Z 1684.732,A 0.000,B 0.000,C 90.000,E1 131.757} C_DIS
LIN {X -0.020,Y -190.080,Z 1684.723,A 0.000,B 0.000,C 90.000,E1 130.135} C_DIS
LIN {X 0.029,Y -195.854,Z 1684.705,A 0.000,B 0.000,C 90.000,E1 126.824} C_DIS
LIN {X -0.062,Y -200.686,Z 1684.691,A 0.000,B 0.000,C 90.000,E1 124.405} C_DIS
LIN {X -0.046,Y -206.571,Z 1684.673,A 0.000,B 0.000,C 90.000,E1 121.180} C_DIS
LIN {X -0.064,Y -208.293,Z 1684.668,A 0.000,B 0.000,C 90.000,E1 120.335} C_DIS
LIN {X -0.152,Y -330.042,Z 1684.668,A 0.000,B 0.000,C 90.000,E1 120.335} C_DIS
LIN {X 0.034,Y -336.146,Z 1684.667,A 0.000,B 0.000,C 90.000,E1 120.129} C_DIS
LIN {X 0.055,Y -338.676,Z 1684.667,A 0.000,B 0.000,C 90.000,E1 119.951} C_DIS
LIN {X -0.096,Y -342.349,Z 1684.664,A 0.000,B 0.000,C 90.000,E1 119.589} C_DIS
LIN {X 0.020,Y -344.248,Z 1684.663,A 0.000,B 0.000,C 90.000,E1 119.283} C_DIS
LIN {X 0.007,Y -345.736,Z 1684.661,A 0.000,B 0.000,C 90.000,E1 118.999} C_DIS
LIN {X -0.114,Y -358.305,Z 1684.646,A 0.000,B 0.000,C 90.000,E1 116.283} C_DIS
LIN {X -0.018,Y -372.359,Z 1684.631,A 0.000,B 0.000,C 90.000,E1 113.590} C_DIS
LIN {X -0.146,Y -386.203,Z 1684.618,A 0.000,B 0.000,C 90.000,E1 111.280} C_DIS
LIN {X 0.147,Y -401.418,Z 1684.605,A 0.000,B 0.000,C 90.000,E1 108.960} C_DIS
LIN {X 0.187,Y -418.111,Z 1684.593,A 0.000,B 0.000,C 90.000,E1 106.732} C_DIS
LIN {X -0.013,Y -436.397,Z 1684.581,A 0.000,B 0.000,C 90.000,E1 104.592} C_DIS
LIN {X -0.190,Y -456.101,Z 1684.569,A 0.000,B 0.000,C 90.000,E1 102.535} C_DIS
LIN {X -0.049,Y -476.422,Z 1684.559,A 0.000,B 0.000,C 90.000,E1 100.602} C_DIS
LIN {X 0.009,Y -499.869,Z 1684.548,A 0.000,B 0.000,C 90.000,E1 98.624} C_DIS
LIN {X 0.162,Y -502.518,Z 1684.547,A 0.000,B 0.000,C 90.000,E1 98.398} C_DIS
LIN {X 0.072,Y -506.390,Z 1684.544,A 0.000,B 0.000,C 90.000,E1 97.992} C_DIS
LIN {X 0.007,Y -507.880,Z 1684.543,A 0.000,B 0.000,C 90.000,E1 97.757} C_DIS
LIN {X -0.127,Y -508.985,Z 1684.542,A 0.000,B 0.000,C 90.000,E1 97.530} C_DIS
LIN {X 0.210,Y -510.264,Z 1684.539,A 0.000,B 0.000,C 90.000,E1 97.011} C_DIS
LIN {X 0.046,Y -510.489,Z 1684.536,A 0.000,B 0.000,C 90.000,E1 96.549} C_DIS
LIN {X -0.110,Y -509.697,Z 1684.534,A 0.000,B 0.000,C 90.000,E1 96.087} C_DIS
LIN {X 0.240,Y -507.747,Z 1684.531,A 0.000,B 0.000,C 90.000,E1 95.568} C_DIS
LIN {X 0.077,Y -504.455,Z 1684.528,A 0.000,B 0.000,C 90.000,E1 95.106} C_DIS
LIN {X -0.065,Y -493.827,Z 1684.520,A 0.000,B 0.000,C 90.000,E1 93.669} C_DIS
LIN {X -0.083,Y -481.329,Z 1684.511,A 0.000,B 0.000,C 90.000,E1 91.949} C_DIS
LIN {X 0.135,Y -468.711,Z 1684.501,A 0.000,B 0.000,C 90.000,E1 90.172} C_DIS
LIN {X -0.157,Y -457.801,Z 1684.493,A 0.000,B 0.000,C 90.000,E1 88.682} C_DIS
LIN {X -0.165,Y -446.705,Z 1684.484,A 0.000,B 0.000,C 90.000,E1 87.135} C_DIS
LIN {X 0.101,Y -435.370,Z 1684.475,A 0.000,B 0.000,C 90.000,E1 85.527} C_DIS
LIN {X -0.108,Y -422.063,Z 1684.465,A 0.000,B 0.000,C 90.000,E1 83.685} C_DIS
LIN {X 0.116,Y -405.452,Z 1684.451,A 0.000,B 0.000,C 90.000,E1 81.197} C_DIS
LIN {X 0.111,Y -384.573,Z 1684.432,A 0.000,B 0.000,C 90.000,E1 77.825} C_DIS
LIN {X 0.081,Y -368.025,Z 1684.416,A 0.000,B 0.000,C 90.000,E1 74.936} C_DIS
LIN {X -0.121,Y -355.233,Z 1684.403,A 0.000,B 0.000,C 90.000,E1 72.598} C_DIS
LIN {X -0.137,Y -337.073,Z 1684.383,A 0.000,B 0.000,C 90.000,E1 68.954} C_DIS
LIN {X 0.119,Y -324.351,Z 1684.367,A 0.000,B 0.000,C 90.000,E1 66.102} C_DIS
LIN {X 0.001,Y -314.712,Z 1684.355,A 0.000,B 0.000,C 90.000,E1 63.896} C_DIS
LIN {X -0.049,Y -305.276,Z 1684.342,A 0.000,B 0.000,C 90.000,E1 61.641} C_DIS
LIN {X -0.008,Y -295.857,Z 1684.330,A 0.000,B 0.000,C 90.000,E1 59.331} C_DIS
LIN {X -0.012,Y -287.558,Z 1684.318,A 0.000,B 0.000,C 90.000,E1 57.327} C_DIS
LIN {X -0.098,Y -279.066,Z 1684.307,A 0.000,B 0.000,C 90.000,E1 55.308} C_DIS
LIN {X 0.044,Y -270.427,Z 1684.296,A 0.000,B 0.000,C 90.000,E1 53.210} C_DIS
LIN {X -0.082,Y -257.690,Z 1684.278,A 0.000,B 0.000,C 90.000,E1 50.070} C_DIS
LIN {X -0.076,Y -245.547,Z 1684.260,A 0.000,B 0.000,C 90.000,E1 46.824} C_DIS
LIN {X -0.040,Y -235.542,Z 1684.244,A 0.000,B 0.000,C 90.000,E1 43.866} C_DIS
LIN {X -0.065,Y -226.411,Z 1684.227,A 0.000,B 0.000,C 90.000,E1 40.862} C_DIS
LIN {X -0.094,Y -218.072,Z 1684.210,A 0.000,B 0.000,C 90.000,E1 37.810} C_DIS
LIN {X -0.071,Y -210.509,Z 1684.193,A 0.000,B 0.000,C 90.000,E1 34.692} C_DIS
LIN {X -0.016,Y -203.590,Z 1684.175,A 0.000,B 0.000,C 90.000,E1 31.514} C_DIS
LIN {X -0.033,Y -197.218,Z 1684.157,A 0.000,B 0.000,C 90.000,E1 28.309} C_DIS
LIN {X 0.055,Y -191.426,Z 1684.139,A 0.000,B 0.000,C 90.000,E1 25.027} C_DIS
LIN {X -0.075,Y -186.142,Z 1684.121,A 0.000,B 0.000,C 90.000,E1 21.770} C_DIS
LIN {X -0.020,Y -181.492,Z 1684.102,A 0.000,B 0.000,C 90.000,E1 18.417} C_DIS
LIN {X 0.094,Y -177.483,Z 1684.083,A 0.000,B 0.000,C 90.000,E1 15.009} C_DIS
LIN {X 0.002,Y -173.504,Z 1684.060,A 0.000,B 0.000,C 90.000,E1 10.782} C_DIS
LIN {X 0.002,Y -169.978,Z 1684.031,A 0.000,B 0.000,C 90.000,E1 5.625} C_DIS
LIN {X -0.031,Y -167.547,Z 1683.997,A 0.000,B 0.000,C 90.000,E1 359.542} C_DIS
LIN {X -0.012,Y -168.380,Z 1683.930,A 0.000,B 0.000,C 90.000,E1 347.353} C_DIS
LIN {X 0.065,Y -170.980,Z 1683.901,A 0.000,B 0.000,C 90.000,E1 342.127} C_DIS
LIN {X -0.018,Y -174.330,Z 1683.877,A 0.000,B 0.000,C 90.000,E1 337.847} C_DIS
LIN {X 0.024,Y -178.969,Z 1683.853,A 0.000,B 0.000,C 90.000,E1 333.563} C_DIS
LIN {X -0.054,Y -183.496,Z 1683.834,A 0.000,B 0.000,C 90.000,E1 330.205} C_DIS
LIN {X 0.024,Y -188.983,Z 1683.816,A 0.000,B 0.000,C 90.000,E1 326.834} C_DIS
LIN {X 0.011,Y -193.805,Z 1683.802,A 0.000,B 0.000,C 90.000,E1 324.356} C_DIS
LIN {X -0.004,Y -199.225,Z 1683.788,A 0.000,B 0.000,C 90.000,E1 321.904} C_DIS
LIN {X -0.058,Y -206.417,Z 1683.773,A 0.000,B 0.000,C 90.000,E1 319.094} C_DIS
LIN {X 0.019,Y -214.634,Z 1683.757,A 0.000,B 0.000,C 90.000,E1 316.296} C_DIS
LIN {X -0.023,Y -223.907,Z 1683.742,A 0.000,B 0.000,C 90.000,E1 313.581} C_DIS
LIN {X -0.016,Y -234.233,Z 1683.727,A 0.000,B 0.000,C 90.000,E1 310.906} C_DIS
LIN {X -0.051,Y -244.209,Z 1683.715,A 0.000,B 0.000,C 90.000,E1 308.669} C_DIS
LIN {X 0.138,Y -253.387,Z 1683.705,A 0.000,B 0.000,C 90.000,E1 306.790} C_DIS
LIN {X -0.182,Y -269.747,Z 1683.689,A 0.000,B 0.000,C 90.000,E1 303.992} C_DIS
LIN {X -0.077,Y -283.150,Z 1683.677,A 0.000,B 0.000,C 90.000,E1 301.878} C_DIS
LIN {X -0.002,Y -299.915,Z 1683.664,A 0.000,B 0.000,C 90.000,E1 299.489} C_DIS
LIN {X 0.046,Y -317.341,Z 1683.651,A 0.000,B 0.000,C 90.000,E1 297.180} C_DIS
LIN {X -0.028,Y -329.861,Z 1683.642,A 0.000,B 0.000,C 90.000,E1 295.591} C_DIS
LIN {X 0.102,Y -347.431,Z 1683.630,A 0.000,B 0.000,C 90.000,E1 293.387} C_DIS
LIN {X -0.074,Y -360.041,Z 1683.622,A 0.000,B 0.000,C 90.000,E1 291.897} C_DIS
LIN {X 0.109,Y -367.429,Z 1683.617,A 0.000,B 0.000,C 90.000,E1 290.972} C_DIS
LIN {X -0.020,Y -376.763,Z 1683.610,A 0.000,B 0.000,C 90.000,E1 289.812} C_DIS
LIN {X 0.192,Y -383.192,Z 1683.605,A 0.000,B 0.000,C 90.000,E1 288.906} C_DIS
LIN {X 0.111,Y -388.909,Z 1683.600,A 0.000,B 0.000,C 90.000,E1 288.055} C_DIS
LIN {X -0.047,Y -393.774,Z 1683.596,A 0.000,B 0.000,C 90.000,E1 287.221} C_DIS
LIN {X 0.168,Y -396.463,Z 1683.593,A 0.000,B 0.000,C 90.000,E1 286.622} C_DIS
LIN {X 0.019,Y -398.753,Z 1683.589,A 0.000,B 0.000,C 90.000,E1 286.079} C_DIS
LIN {X -0.119,Y -400.672,Z 1683.586,A 0.000,B 0.000,C 90.000,E1 285.536} C_DIS
LIN {X 0.029,Y -402.256,Z 1683.583,A 0.000,B 0.000,C 90.000,E1 284.954} C_DIS
LIN {X -0.095,Y -403.505,Z 1683.580,A 0.000,B 0.000,C 90.000,E1 284.411} C_DIS
LIN {X 0.079,Y -404.293,Z 1683.577,A 0.000,B 0.000,C 90.000,E1 283.828} C_DIS
LIN {X -0.128,Y -404.739,Z 1683.574,A 0.000,B 0.000,C 90.000,E1 283.300} C_DIS
LIN {X 0.066,Y -404.707,Z 1683.571,A 0.000,B 0.000,C 90.000,E1 282.715} C_DIS
LIN {X -0.047,Y -404.235,Z 1683.568,A 0.000,B 0.000,C 90.000,E1 282.175} C_DIS
LIN {X 0.147,Y -403.217,Z 1683.564,A 0.000,B 0.000,C 90.000,E1 281.591} C_DIS
LIN {X -0.134,Y -401.749,Z 1683.561,A 0.000,B 0.000,C 90.000,E1 281.074} C_DIS
LIN {X 0.053,Y -399.731,Z 1683.558,A 0.000,B 0.000,C 90.000,E1 280.489} C_DIS
LIN {X -0.164,Y -397.221,Z 1683.555,A 0.000,B 0.000,C 90.000,E1 279.962} C_DIS
LIN {X -0.006,Y -392.542,Z 1683.551,A 0.000,B 0.000,C 90.000,E1 279.095} C_DIS
LIN {X 0.173,Y -387.074,Z 1683.546,A 0.000,B 0.000,C 90.000,E1 278.219} C_DIS
LIN {X -0.142,Y -380.957,Z 1683.541,A 0.000,B 0.000,C 90.000,E1 277.409} C_DIS
LIN {X -0.140,Y -376.316,Z 1683.538,A 0.000,B 0.000,C 90.000,E1 276.834} C_DIS
LIN {X -0.163,Y -371.063,Z 1683.535,A 0.000,B 0.000,C 90.000,E1 276.258} C_DIS
LIN {X -0.047,Y -365.353,Z 1683.531,A 0.000,B 0.000,C 90.000,E1 275.682} C_DIS
LIN {X -0.019,Y -359.396,Z 1683.529,A 0.000,B 0.000,C 90.000,E1 275.163} C_DIS
LIN {X -0.106,Y -353.239,Z 1683.526,A 0.000,B 0.000,C 90.000,E1 274.702} C_DIS
LIN {X 0.060,Y -346.790,Z 1683.524,A 0.000,B 0.000,C 90.000,E1 274.245} C_DIS
LIN {X 0.151,Y -336.968,Z 1683.521,A 0.000,B 0.000,C 90.000,E1 273.669} C_DIS
LIN {X -0.142,Y -330.370,Z 1683.519,A 0.000,B 0.000,C 90.000,E1 273.383} C_DIS
LIN {X -0.112,Y -320.333,Z 1683.516,A 0.000,B 0.000,C 90.000,E1 272.922} C_DIS
LIN {X -0.049,Y -313.622,Z 1683.515,A 0.000,B 0.000,C 90.000,E1 272.636} C_DIS
LIN {X -0.138,Y -306.968,Z 1683.513,A 0.000,B 0.000,C 90.000,E1 272.407} C_DIS
LIN {X -0.014,Y -296.834,Z 1683.511,A 0.000,B 0.000,C 90.000,E1 272.064} C_DIS
LIN {X 0.076,Y -285.934,Z 1683.510,A 0.000,B 0.000,C 90.000,E1 271.776} C_DIS
LIN {X -0.108,Y -278.011,Z 1683.509,A 0.000,B 0.000,C 90.000,E1 271.661} C_DIS
LIN {X 0.094,Y -269.130,Z 1683.508,A 0.000,B 0.000,C 90.000,E1 271.489} C_DIS
LIN {X -0.055,Y -256.501,Z 1683.508,A 0.000,B 0.000,C 90.000,E1 271.432} C_DIS
LIN {X 0.035,Y -231.026,Z 1683.508,A 0.000,B 0.000,C 90.000,E1 271.375} C_DIS
LIN {X 0.010,Y -223.918,Z 1683.508,A 0.000,B 0.000,C 90.000,E1 271.375} C_DIS
LIN {X -0.026,Y -196.361,Z 1683.507,A 0.000,B 0.000,C 90.000,E1 271.318} C_DIS
LIN {X -0.035,Y -184.496,Z 1683.507,A 0.000,B 0.000,C 90.000,E1 271.260} C_DIS
LIN {X -0.066,Y -181.403,Z 1683.507,A 0.000,B 0.000,C 90.000,E1 271.260} C_DIS
LIN {X -0.025,Y -181.580,Z 1683.501,A 0.000,B 0.000,C 90.000,E1 270.229} C_DIS
LIN {X -0.021,Y -180.862,Z 1683.472,A 0.000,B 0.000,C 90.000,E1 265.008} C_DIS
LIN {X 0.033,Y -178.976,Z 1683.444,A 0.000,B 0.000,C 90.000,E1 259.926} C_DIS
LIN {X 0.042,Y -177.939,Z 1683.435,A 0.000,B 0.000,C 90.000,E1 258.229} C_DIS
LIN {X 0.057,Y -175.578,Z 1683.411,A 0.000,B 0.000,C 90.000,E1 253.976} C_DIS
LIN {X 0.063,Y -172.305,Z 1683.387,A 0.000,B 0.000,C 90.000,E1 249.699} C_DIS
LIN {X 0.041,Y -171.783,Z 1683.383,A 0.000,B 0.000,C 90.000,E1 248.847} C_DIS
LIN {X -0.081,Y -169.449,Z 1683.368,A 0.000,B 0.000,C 90.000,E1 246.305} C_DIS
LIN {X -0.025,Y -166.779,Z 1683.349,A 0.000,B 0.000,C 90.000,E1 242.820} C_DIS
LIN {X -0.029,Y -162.760,Z 1683.325,A 0.000,B 0.000,C 90.000,E1 238.456} C_DIS
LIN {X -0.053,Y -161.450,Z 1683.315,A 0.000,B 0.000,C 90.000,E1 236.707} C_DIS
LIN {X -0.011,Y -157.443,Z 1683.290,A 0.000,B 0.000,C 90.000,E1 232.271} C_DIS
LIN {X 0.023,Y -155.451,Z 1683.276,A 0.000,B 0.000,C 90.000,E1 229.585} C_DIS
LIN {X 0.072,Y -151.769,Z 1683.251,A 0.000,B 0.000,C 90.000,E1 225.081} C_DIS
LIN {X -0.019,Y -149.972,Z 1683.236,A 0.000,B 0.000,C 90.000,E1 222.405} C_DIS
LIN {X -0.007,Y -146.809,Z 1683.210,A 0.000,B 0.000,C 90.000,E1 217.855} C_DIS
LIN {X 0.009,Y -145.387,Z 1683.195,A 0.000,B 0.000,C 90.000,E1 215.105} C_DIS
LIN {X 0.001,Y -142.444,Z 1683.164,A 0.000,B 0.000,C 90.000,E1 209.589} C_DIS
LIN {X -0.017,Y -141.437,Z 1683.149,A 0.000,B 0.000,C 90.000,E1 206.821} C_DIS
LIN {X 0.028,Y -139.367,Z 1683.113,A 0.000,B 0.000,C 90.000,E1 200.301} C_DIS
LIN {X 0.015,Y -138.813,Z 1683.097,A 0.000,B 0.000,C 90.000,E1 197.511} C_DIS
LIN {X 0.066,Y -138.352,Z 1683.056,A 0.000,B 0.000,C 90.000,E1 190.018} C_DIS
LIN {X 0.042,Y -139.539,Z 1683.004,A 0.000,B 0.000,C 90.000,E1 180.688} C_DIS
LIN {X -0.006,Y -141.231,Z 1682.973,A 0.000,B 0.000,C 90.000,E1 175.122} C_DIS
LIN {X -0.047,Y -142.602,Z 1682.957,A 0.000,B 0.000,C 90.000,E1 172.356} C_DIS
LIN {X 0.048,Y -144.911,Z 1682.932,A 0.000,B 0.000,C 90.000,E1 167.701} C_DIS
LIN {X 0.041,Y -147.539,Z 1682.911,A 0.000,B 0.000,C 90.000,E1 164.031} C_DIS
LIN {X -0.068,Y -150.139,Z 1682.891,A 0.000,B 0.000,C 90.000,E1 160.423} C_DIS
LIN {X -0.057,Y -153.505,Z 1682.871,A 0.000,B 0.000,C 90.000,E1 156.794} C_DIS
LIN {X 0.005,Y -157.871,Z 1682.846,A 0.000,B 0.000,C 90.000,E1 152.281} C_DIS
LIN {X -0.040,Y -162.158,Z 1682.826,A 0.000,B 0.000,C 90.000,E1 148.742} C_DIS
LIN {X 0.075,Y -166.364,Z 1682.807,A 0.000,B 0.000,C 90.000,E1 145.182} C_DIS
LIN {X -0.056,Y -171.380,Z 1682.787,A 0.000,B 0.000,C 90.000,E1 141.743} C_DIS
LIN {X -0.014,Y -176.290,Z 1682.768,A 0.000,B 0.000,C 90.000,E1 138.286} C_DIS
LIN {X -0.013,Y -180.576,Z 1682.754,A 0.000,B 0.000,C 90.000,E1 135.729} C_DIS
LIN {X -0.034,Y -185.978,Z 1682.735,A 0.000,B 0.000,C 90.000,E1 132.366} C_DIS
LIN {X 0.022,Y -190.610,Z 1682.721,A 0.000,B 0.000,C 90.000,E1 129.850} C_DIS
LIN {X -0.071,Y -196.360,Z 1682.703,A 0.000,B 0.000,C 90.000,E1 126.583} C_DIS
LIN {X 0.005,Y -201.154,Z 1682.690,A 0.000,B 0.000,C 90.000,E1 124.119} C_DIS
LIN {X 0.015,Y -207.463,Z 1682.671,A 0.000,B 0.000,C 90.000,E1 120.718} C_DIS
LIN {X 0.045,Y -208.231,Z 1682.669,A 0.000,B 0.000,C 90.000,E1 120.335} C_DIS
LIN {X 0.032,Y -330.483,Z 1682.669,A 0.000,B 0.000,C 90.000,E1 120.335} C_DIS
LIN {X 0.093,Y -334.922,Z 1682.668,A 0.000,B 0.000,C 90.000,E1 120.207} C_DIS
LIN {X -0.135,Y -337.016,Z 1682.667,A 0.000,B 0.000,C 90.000,E1 120.129} C_DIS
LIN {X 0.119,Y -340.887,Z 1682.665,A 0.000,B 0.000,C 90.000,E1 119.745} C_DIS
LIN {X -0.105,Y -344.394,Z 1682.663,A 0.000,B 0.000,C 90.000,E1 119.283} C_DIS
LIN {X 0.207,Y -347.247,Z 1682.659,A 0.000,B 0.000,C 90.000,E1 118.615} C_DIS
LIN {X -0.018,Y -359.984,Z 1682.644,A 0.000,B 0.000,C 90.000,E1 115.924} C_DIS
LIN {X -0.052,Y -374.235,Z 1682.629,A 0.000,B 0.000,C 90.000,E1 113.259} C_DIS
LIN {X 0.075,Y -388.269,Z 1682.616,A 0.000,B 0.000,C 90.000,E1 110.918} C_DIS
LIN {X -0.078,Y -403.690,Z 1682.604,A 0.000,B 0.000,C 90.000,E1 108.671} C_DIS
LIN {X 0.018,Y -420.604,Z 1682.591,A 0.000,B 0.000,C 90.000,E1 106.441} C_DIS
LIN {X -0.122,Y -439.127,Z 1682.579,A 0.000,B 0.000,C 90.000,E1 104.300} C_DIS
LIN {X -0.134,Y -458.957,Z 1682.568,A 0.000,B 0.000,C 90.000,E1 102.243} C_DIS
LIN {X 0.201,Y -479.355,Z 1682.557,A 0.000,B 0.000,C 90.000,E1 100.310} C_DIS
LIN {X -0.101,Y -502.829,Z 1682.547,A 0.000,B 0.000,C 90.000,E1 98.398} C_DIS
LIN {X 0.148,Y -504.886,Z 1682.545,A 0.000,B 0.000,C 90.000,E1 98.163} C_DIS
LIN {X 0.026,Y -506.693,Z 1682.544,A 0.000,B 0.000,C 90.000,E1 97.936} C_DIS
LIN {X -0.028,Y -508.045,Z 1682.543,A 0.000,B 0.000,C 90.000,E1 97.701} C_DIS
LIN {X -0.206,Y -509.733,Z 1682.540,A 0.000,B 0.000,C 90.000,E1 97.239} C_DIS
LIN {X 0.130,Y -510.311,Z 1682.537,A 0.000,B 0.000,C 90.000,E1 96.720} C_DIS
LIN {X -0.031,Y -509.877,Z 1682.535,A 0.000,B 0.000,C 90.000,E1 96.258} C_DIS
LIN {X -0.188,Y -508.359,Z 1682.532,A 0.000,B 0.000,C 90.000,E1 95.796} C_DIS
LIN {X 0.211,Y -507.109,Z 1682.531,A 0.000,B 0.000,C 90.000,E1 95.511} C_DIS
LIN {X 0.238,Y -498.448,Z 1682.524,A 0.000,B 0.000,C 90.000,E1 94.302} C_DIS
LIN {X -0.157,Y -485.965,Z 1682.515,A 0.000,B 0.000,C 90.000,E1 92.636} C_DIS
LIN {X 0.152,Y -473.410,Z 1682.505,A 0.000,B 0.000,C 90.000,E1 90.859} C_DIS
LIN {X 0.190,Y -460.736,Z 1682.495,A 0.000,B 0.000,C 90.000,E1 89.083} C_DIS
LIN {X 0.226,Y -449.683,Z 1682.486,A 0.000,B 0.000,C 90.000,E1 87.535} C_DIS
LIN {X 0.071,Y -438.376,Z 1682.478,A 0.000,B 0.000,C 90.000,E1 85.988} C_DIS
LIN {X -0.077,Y -425.077,Z 1682.467,A 0.000,B 0.000,C 90.000,E1 84.147} C_DIS
LIN {X -0.126,Y -406.478,Z 1682.452,A 0.000,B 0.000,C 90.000,E1 81.432} C_DIS
LIN {X -0.011,Y -385.486,Z 1682.434,A 0.000,B 0.000,C 90.000,E1 78.049} C_DIS
LIN {X -0.084,Y -370.486,Z 1682.419,A 0.000,B 0.000,C 90.000,E1 75.463} C_DIS
LIN {X 0.020,Y -357.608,Z 1682.406,A 0.000,B 0.000,C 90.000,E1 73.087} C_DIS
LIN {X 0.067,Y -340.704,Z 1682.388,A 0.000,B 0.000,C 90.000,E1 69.752} C_DIS
LIN {X 0.016,Y -329.230,Z 1682.374,A 0.000,B 0.000,C 90.000,E1 67.283} C_DIS
LIN {X -0.184,Y -318.153,Z 1682.360,A 0.000,B 0.000,C 90.000,E1 64.793} C_DIS
LIN {X 0.063,Y -305.961,Z 1682.344,A 0.000,B 0.000,C 90.000,E1 61.847} C_DIS
LIN {X 0.113,Y -296.515,Z 1682.331,A 0.000,B 0.000,C 90.000,E1 59.537} C_DIS
LIN {X -0.127,Y -288.216,Z 1682.320,A 0.000,B 0.000,C 90.000,E1 57.582} C_DIS
LIN {X 0.038,Y -279.731,Z 1682.308,A 0.000,B 0.000,C 90.000,E1 55.515} C_DIS
LIN {X -0.101,Y -269.638,Z 1682.295,A 0.000,B 0.000,C 90.000,E1 53.130} C_DIS
LIN {X 0.128,Y -256.925,Z 1682.277,A 0.000,B 0.000,C 90.000,E1 49.908} C_DIS
LIN {X -0.067,Y -244.865,Z 1682.259,A 0.000,B 0.000,C 90.000,E1 46.701} C_DIS
LIN {X 0.113,Y -234.932,Z 1682.243,A 0.000,B 0.000,C 90.000,E1 43.704} C_DIS
LIN {X 0.014,Y -224.798,Z 1682.224,A 0.000,B 0.000,C 90.000,E1 40.334} C_DIS
LIN {X -0.053,Y -216.639,Z 1682.207,A 0.000,B 0.000,C 90.000,E1 37.282} C_DIS
LIN {X 0.098,Y -209.229,Z 1682.190,A 0.000,B 0.000,C 90.000,E1 34.119} C_DIS
LIN {X -0.101,Y -202.424,Z 1682.172,A 0.000,B 0.000,C 90.000,E1 31.003} C_DIS
LIN {X -0.045,Y -196.123,Z 1682.154,A 0.000,B 0.000,C 90.000,E1 27.769} C_DIS
LIN {X 0.093,Y -189.056,Z 1682.131,A 0.000,B 0.000,C 90.000,E1 23.643} C_DIS
LIN {X 0.003,Y -184.050,Z 1682.113,A 0.000,B 0.000,C 90.000,E1 20.355} C_DIS
LIN {X 0.061,Y -179.630,Z 1682.094,A 0.000,B 0.000,C 90.000,E1 16.985} C_DIS
LIN {X 0.083,Y -175.956,Z 1682.076,A 0.000,B 0.000,C 90.000,E1 13.592} C_DIS
LIN {X 0.080,Y -172.332,Z 1682.052,A 0.000,B 0.000,C 90.000,E1 9.321} C_DIS
LIN {X -0.029,Y -169.174,Z 1682.023,A 0.000,B 0.000,C 90.000,E1 4.188} C_DIS
LIN {X 0.081,Y -167.213,Z 1681.988,A 0.000,B 0.000,C 90.000,E1 357.764} C_DIS
LIN {X -0.015,Y -168.366,Z 1681.930,A 0.000,B 0.000,C 90.000,E1 347.353} C_DIS
LIN {X 0.063,Y -170.982,Z 1681.901,A 0.000,B 0.000,C 90.000,E1 342.127} C_DIS
LIN {X -0.020,Y -174.356,Z 1681.877,A 0.000,B 0.000,C 90.000,E1 337.847} C_DIS
LIN {X 0.039,Y -178.017,Z 1681.858,A 0.000,B 0.000,C 90.000,E1 334.409} C_DIS
LIN {X -0.064,Y -182.354,Z 1681.839,A 0.000,B 0.000,C 90.000,E1 331.051} C_DIS
LIN {X 0.047,Y -187.623,Z 1681.820,A 0.000,B 0.000,C 90.000,E1 327.661} C_DIS
LIN {X 0.011,Y -192.240,Z 1681.807,A 0.000,B 0.000,C 90.000,E1 325.182} C_DIS
LIN {X 0.009,Y -197.478,Z 1681.793,A 0.000,B 0.000,C 90.000,E1 322.718} C_DIS
LIN {X -0.091,Y -204.440,Z 1681.777,A 0.000,B 0.000,C 90.000,E1 319.908} C_DIS
LIN {X 0.098,Y -212.350,Z 1681.762,A 0.000,B 0.000,C 90.000,E1 317.067} C_DIS
LIN {X 0.007,Y -221.354,Z 1681.746,A 0.000,B 0.000,C 90.000,E1 314.352} C_DIS
LIN {X -0.044,Y -231.363,Z 1681.731,A 0.000,B 0.000,C 90.000,E1 311.676} C_DIS
LIN {X 0.019,Y -240.949,Z 1681.719,A 0.000,B 0.000,C 90.000,E1 309.402} C_DIS
LIN {X 0.159,Y -251.646,Z 1681.707,A 0.000,B 0.000,C 90.000,E1 307.156} C_DIS
LIN {X -0.051,Y -267.743,Z 1681.691,A 0.000,B 0.000,C 90.000,E1 304.326} C_DIS
LIN {X -0.032,Y -283.259,Z 1681.677,A 0.000,B 0.000,C 90.000,E1 301.878} C_DIS
LIN {X 0.048,Y -300.005,Z 1681.664,A 0.000,B 0.000,C 90.000,E1 299.489} C_DIS
LIN {X -0.044,Y -317.424,Z 1681.651,A 0.000,B 0.000,C 90.000,E1 297.206} C_DIS
LIN {X 0.031,Y -329.932,Z 1681.642,A 0.000,B 0.000,C 90.000,E1 295.591} C_DIS
LIN {X 0.177,Y -347.443,Z 1681.630,A 0.000,B 0.000,C 90.000,E1 293.387} C_DIS
LIN {X -0.006,Y -360.027,Z 1681.622,A 0.000,B 0.000,C 90.000,E1 291.897} C_DIS
LIN {X -0.226,Y -369.780,Z 1681.615,A 0.000,B 0.000,C 90.000,E1 290.737} C_DIS
LIN {X 0.050,Y -376.742,Z 1681.610,A 0.000,B 0.000,C 90.000,E1 289.812} C_DIS
LIN {X -0.099,Y -383.175,Z 1681.605,A 0.000,B 0.000,C 90.000,E1 288.960} C_DIS
LIN {X 0.183,Y -388.886,Z 1681.600,A 0.000,B 0.000,C 90.000,E1 288.055} C_DIS
LIN {X 0.025,Y -393.786,Z 1681.596,A 0.000,B 0.000,C 90.000,E1 287.221} C_DIS
LIN {X -0.139,Y -396.517,Z 1681.593,A 0.000,B 0.000,C 90.000,E1 286.677} C_DIS
LIN {X 0.093,Y -398.815,Z 1681.589,A 0.000,B 0.000,C 90.000,E1 286.079} C_DIS
LIN {X -0.153,Y -400.760,Z 1681.586,A 0.000,B 0.000,C 90.000,E1 285.552} C_DIS
LIN {X 0.104,Y -402.360,Z 1681.583,A 0.000,B 0.000,C 90.000,E1 284.954} C_DIS
LIN {X -0.019,Y -403.599,Z 1681.580,A 0.000,B 0.000,C 90.000,E1 284.411} C_DIS
LIN {X 0.157,Y -404.451,Z 1681.577,A 0.000,B 0.000,C 90.000,E1 283.828} C_DIS
LIN {X -0.050,Y -404.886,Z 1681.574,A 0.000,B 0.000,C 90.000,E1 283.300} C_DIS
LIN {X 0.145,Y -404.907,Z 1681.571,A 0.000,B 0.000,C 90.000,E1 282.715} C_DIS
LIN {X -0.053,Y -404.412,Z 1681.568,A 0.000,B 0.000,C 90.000,E1 282.187} C_DIS
LIN {X 0.145,Y -403.480,Z 1681.565,A 0.000,B 0.000,C 90.000,E1 281.602} C_DIS
LIN {X -0.054,Y -402.018,Z 1681.562,A 0.000,B 0.000,C 90.000,E1 281.074} C_DIS
LIN {X 0.134,Y -400.015,Z 1681.558,A 0.000,B 0.000,C 90.000,E1 280.489} C_DIS
LIN {X -0.081,Y -397.487,Z 1681.555,A 0.000,B 0.000,C 90.000,E1 279.962} C_DIS
LIN {X 0.078,Y -392.774,Z 1681.551,A 0.000,B 0.000,C 90.000,E1 279.095} C_DIS
LIN {X -0.125,Y -387.301,Z 1681.546,A 0.000,B 0.000,C 90.000,E1 278.276} C_DIS
LIN {X -0.056,Y -381.142,Z 1681.541,A 0.000,B 0.000,C 90.000,E1 277.409} C_DIS
LIN {X -0.054,Y -376.468,Z 1681.538,A 0.000,B 0.000,C 90.000,E1 276.834} C_DIS
LIN {X -0.061,Y -371.215,Z 1681.535,A 0.000,B 0.000,C 90.000,E1 276.258} C_DIS
LIN {X 0.086,Y -365.499,Z 1681.532,A 0.000,B 0.000,C 90.000,E1 275.682} C_DIS
LIN {X 0.134,Y -359.559,Z 1681.529,A 0.000,B 0.000,C 90.000,E1 275.163} C_DIS
LIN {X 0.060,Y -353.372,Z 1681.526,A 0.000,B 0.000,C 90.000,E1 274.702} C_DIS
LIN {X -0.115,Y -346.940,Z 1681.524,A 0.000,B 0.000,C 90.000,E1 274.302} C_DIS
LIN {X -0.024,Y -337.068,Z 1681.521,A 0.000,B 0.000,C 90.000,E1 273.726} C_DIS
LIN {X 0.126,Y -327.167,Z 1681.518,A 0.000,B 0.000,C 90.000,E1 273.212} C_DIS
LIN {X -0.069,Y -317.214,Z 1681.516,A 0.000,B 0.000,C 90.000,E1 272.808} C_DIS
LIN {X 0.042,Y -307.278,Z 1681.513,A 0.000,B 0.000,C 90.000,E1 272.407} C_DIS
LIN {X 0.130,Y -297.078,Z 1681.512,A 0.000,B 0.000,C 90.000,E1 272.064} C_DIS
LIN {X 0.032,Y -289.871,Z 1681.510,A 0.000,B 0.000,C 90.000,E1 271.892} C_DIS
LIN {X 0.015,Y -278.112,Z 1681.509,A 0.000,B 0.000,C 90.000,E1 271.661} C_DIS
LIN {X -0.052,Y -269.250,Z 1681.509,A 0.000,B 0.000,C 90.000,E1 271.547} C_DIS
LIN {X 0.093,Y -257.956,Z 1681.508,A 0.000,B 0.000,C 90.000,E1 271.432} C_DIS
LIN {X -0.087,Y -236.431,Z 1681.508,A 0.000,B 0.000,C 90.000,E1 271.432} C_DIS
LIN {X -0.107,Y -227.227,Z 1681.508,A 0.000,B 0.000,C 90.000,E1 271.432} C_DIS
LIN {X -0.062,Y -192.042,Z 1681.507,A 0.000,B 0.000,C 90.000,E1 271.318} C_DIS
LIN {X -0.007,Y -184.265,Z 1681.507,A 0.000,B 0.000,C 90.000,E1 271.260} C_DIS
LIN {X -0.039,Y -181.402,Z 1681.507,A 0.000,B 0.000,C 90.000,E1 271.260} C_DIS
LIN {X 0.002,Y -181.580,Z 1681.501,A 0.000,B 0.000,C 90.000,E1 270.229} C_DIS
LIN {X 0.005,Y -180.864,Z 1681.472,A 0.000,B 0.000,C 90.000,E1 265.008} C_DIS
LIN {X 0.059,Y -178.978,Z 1681.444,A 0.000,B 0.000,C 90.000,E1 259.926} C_DIS
LIN {X 0.069,Y -177.945,Z 1681.435,A 0.000,B 0.000,C 90.000,E1 258.229} C_DIS
LIN {X 0.083,Y -175.585,Z 1681.411,A 0.000,B 0.000,C 90.000,E1 253.976} C_DIS
LIN {X -0.072,Y -172.311,Z 1681.387,A 0.000,B 0.000,C 90.000,E1 249.752} C_DIS
LIN {X -0.093,Y -171.788,Z 1681.383,A 0.000,B 0.000,C 90.000,E1 248.901} C_DIS
LIN {X -0.055,Y -169.457,Z 1681.368,A 0.000,B 0.000,C 90.000,E1 246.305} C_DIS
LIN {X 0.000,Y -166.787,Z 1681.349,A 0.000,B 0.000,C 90.000,E1 242.820} C_DIS
LIN {X -0.004,Y -162.766,Z 1681.325,A 0.000,B 0.000,C 90.000,E1 238.456} C_DIS
LIN {X -0.028,Y -161.456,Z 1681.315,A 0.000,B 0.000,C 90.000,E1 236.707} C_DIS
LIN {X 0.013,Y -157.450,Z 1681.290,A 0.000,B 0.000,C 90.000,E1 232.271} C_DIS
LIN {X -0.054,Y -155.460,Z 1681.276,A 0.000,B 0.000,C 90.000,E1 229.622} C_DIS
LIN {X -0.012,Y -151.775,Z 1681.251,A 0.000,B 0.000,C 90.000,E1 225.121} C_DIS
LIN {X 0.005,Y -149.979,Z 1681.236,A 0.000,B 0.000,C 90.000,E1 222.405} C_DIS
LIN {X -0.074,Y -146.815,Z 1681.210,A 0.000,B 0.000,C 90.000,E1 217.890} C_DIS
LIN {X 0.033,Y -145.392,Z 1681.195,A 0.000,B 0.000,C 90.000,E1 215.105} C_DIS
LIN {X -0.050,Y -142.829,Z 1681.170,A 0.000,B 0.000,C 90.000,E1 210.541} C_DIS
LIN {X 0.007,Y -141.441,Z 1681.149,A 0.000,B 0.000,C 90.000,E1 206.821} C_DIS
LIN {X 0.052,Y -139.368,Z 1681.113,A 0.000,B 0.000,C 90.000,E1 200.301} C_DIS
LIN {X 0.037,Y -138.816,Z 1681.097,A 0.000,B 0.000,C 90.000,E1 197.511} C_DIS
LIN {X -0.048,Y -138.352,Z 1681.056,A 0.000,B 0.000,C 90.000,E1 190.074} C_DIS
LIN {X 0.064,Y -139.537,Z 1681.004,A 0.000,B 0.000,C 90.000,E1 180.688} C_DIS
LIN {X 0.017,Y -141.227,Z 1680.973,A 0.000,B 0.000,C 90.000,E1 175.122} C_DIS
LIN {X -0.024,Y -142.599,Z 1680.958,A 0.000,B 0.000,C 90.000,E1 172.356} C_DIS
LIN {X 0.071,Y -144.904,Z 1680.932,A 0.000,B 0.000,C 90.000,E1 167.701} C_DIS
LIN {X 0.024,Y -147.533,Z 1680.911,A 0.000,B 0.000,C 90.000,E1 164.047} C_DIS
LIN {X -0.044,Y -150.131,Z 1680.891,A 0.000,B 0.000,C 90.000,E1 160.423} C_DIS
LIN {X -0.034,Y -153.496,Z 1680.871,A 0.000,B 0.000,C 90.000,E1 156.794} C_DIS
LIN {X 0.030,Y -157.861,Z 1680.846,A 0.000,B 0.000,C 90.000,E1 152.281} C_DIS
LIN {X -0.015,Y -162.147,Z 1680.826,A 0.000,B 0.000,C 90.000,E1 148.742} C_DIS
LIN {X -0.036,Y -166.352,Z 1680.807,A 0.000,B 0.000,C 90.000,E1 145.229} C_DIS
LIN {X -0.031,Y -171.369,Z 1680.787,A 0.000,B 0.000,C 90.000,E1 141.743} C_DIS
LIN {X -0.104,Y -176.277,Z 1680.768,A 0.000,B 0.000,C 90.000,E1 138.324} C_DIS
LIN {X 0.015,Y -180.561,Z 1680.754,A 0.000,B 0.000,C 90.000,E1 135.729} C_DIS
LIN {X -0.007,Y -185.963,Z 1680.735,A 0.000,B 0.000,C 90.000,E1 132.366} C_DIS
LIN {X 0.049,Y -190.595,Z 1680.721,A 0.000,B 0.000,C 90.000,E1 129.850} C_DIS
LIN {X -0.044,Y -196.345,Z 1680.703,A 0.000,B 0.000,C 90.000,E1 126.583} C_DIS
LIN {X 0.033,Y -201.140,Z 1680.690,A 0.000,B 0.000,C 90.000,E1 124.119} C_DIS
LIN {X 0.044,Y -207.446,Z 1680.671,A 0.000,B 0.000,C 90.000,E1 120.718} C_DIS
LIN {X -0.003,Y -208.156,Z 1680.669,A 0.000,B 0.000,C 90.000,E1 120.384} C_DIS
LIN {X -0.048,Y -330.213,Z 1680.669,A 0.000,B 0.000,C 90.000,E1 120.384} C_DIS
LIN {X -0.068,Y -335.028,Z 1680.668,A 0.000,B 0.000,C 90.000,E1 120.256} C_DIS
LIN {X -0.089,Y -337.239,Z 1680.667,A 0.000,B 0.000,C 90.000,E1 120.129} C_DIS
LIN {X 0.060,Y -341.104,Z 1680.665,A 0.000,B 0.000,C 90.000,E1 119.745} C_DIS
LIN {X 0.180,Y -344.578,Z 1680.662,A 0.000,B 0.000,C 90.000,E1 119.205} C_DIS
LIN {X -0.049,Y -360.111,Z 1680.644,A 0.000,B 0.000,C 90.000,E1 115.899} C_DIS
LIN {X 0.100,Y -374.380,Z 1680.629,A 0.000,B 0.000,C 90.000,E1 113.206} C_DIS
LIN {X -0.120,Y -388.430,Z 1680.616,A 0.000,B 0.000,C 90.000,E1 110.918} C_DIS
LIN {X 0.234,Y -403.869,Z 1680.604,A 0.000,B 0.000,C 90.000,E1 108.598} C_DIS
LIN {X -0.185,Y -420.801,Z 1680.591,A 0.000,B 0.000,C 90.000,E1 106.441} C_DIS
LIN {X 0.097,Y -439.345,Z 1680.579,A 0.000,B 0.000,C 90.000,E1 104.245} C_DIS
LIN {X 0.112,Y -459.187,Z 1680.568,A 0.000,B 0.000,C 90.000,E1 102.187} C_DIS
LIN {X 0.005,Y -479.591,Z 1680.557,A 0.000,B 0.000,C 90.000,E1 100.310} C_DIS
LIN {X 0.209,Y -503.014,Z 1680.547,A 0.000,B 0.000,C 90.000,E1 98.341} C_DIS
LIN {X -0.038,Y -504.972,Z 1680.545,A 0.000,B 0.000,C 90.000,E1 98.163} C_DIS
LIN {X -0.173,Y -506.710,Z 1680.544,A 0.000,B 0.000,C 90.000,E1 97.936} C_DIS
LIN {X -0.237,Y -508.010,Z 1680.543,A 0.000,B 0.000,C 90.000,E1 97.701} C_DIS
LIN {X 0.090,Y -509.603,Z 1680.540,A 0.000,B 0.000,C 90.000,E1 97.182} C_DIS
LIN {X -0.080,Y -510.104,Z 1680.537,A 0.000,B 0.000,C 90.000,E1 96.720} C_DIS
LIN {X -0.241,Y -509.591,Z 1680.535,A 0.000,B 0.000,C 90.000,E1 96.258} C_DIS
LIN {X 0.106,Y -507.982,Z 1680.532,A 0.000,B 0.000,C 90.000,E1 95.739} C_DIS
LIN {X 0.000,Y -506.674,Z 1680.531,A 0.000,B 0.000,C 90.000,E1 95.511} C_DIS
LIN {X -0.101,Y -496.201,Z 1680.523,A 0.000,B 0.000,C 90.000,E1 94.073} C_DIS
LIN {X -0.040,Y -483.740,Z 1680.513,A 0.000,B 0.000,C 90.000,E1 92.350} C_DIS
LIN {X -0.068,Y -472.955,Z 1680.505,A 0.000,B 0.000,C 90.000,E1 90.859} C_DIS
LIN {X 0.178,Y -462.105,Z 1680.496,A 0.000,B 0.000,C 90.000,E1 89.312} C_DIS
LIN {X -0.212,Y -451.092,Z 1680.488,A 0.000,B 0.000,C 90.000,E1 87.822} C_DIS
LIN {X 0.110,Y -439.821,Z 1680.479,A 0.000,B 0.000,C 90.000,E1 86.216} C_DIS
LIN {X -0.011,Y -426.481,Z 1680.469,A 0.000,B 0.000,C 90.000,E1 84.375} C_DIS
LIN {X -0.133,Y -409.622,Z 1680.455,A 0.000,B 0.000,C 90.000,E1 81.951} C_DIS
LIN {X 0.024,Y -388.374,Z 1680.437,A 0.000,B 0.000,C 90.000,E1 78.578} C_DIS
LIN {X 0.027,Y -373.238,Z 1680.422,A 0.000,B 0.000,C 90.000,E1 75.992} C_DIS
